SPLINE
SPL {X  -162.820, Y  +574.443, Z    +0.000, E1   +42.333, E3 +366187.799}
SPL {X  -162.820, Y  +568.554, Z    +0.000, E1   +42.362, E3 +366201.161}
SPL {X  -162.820, Y  +561.474, Z    +0.000, E1   +42.369, E3 +366217.346}
SPL {X  -162.820, Y  +555.861, Z    +0.000, E1   +42.349, E3 +366230.151}
SPL {X  -162.820, Y  +550.633, Z    +0.000, E1   +42.421, E3 +366241.681}
SPL {X  -162.820, Y  +546.534, Z    +0.000, E1   +42.268, E3 +366251.890}
SPL {X  -162.820, Y  +539.632, Z    +0.000, E1   +42.488, E3 +366266.611}
SPL {X  -162.820, Y  +533.959, Z    +0.000, E1   +42.310, E3 +366280.308}
SPL {X  -162.820, Y  +527.661, Z    +0.000, E1   +42.425, E3 +366294.304}
SPL {X  -162.820, Y  +521.246, Z    +0.000, E1   +42.365, E3 +366309.057}
SPL {X  -162.820, Y  +515.708, Z    +0.000, E1   +42.333, E3 +366322.019}
SPL {X  -162.820, Y  +510.265, Z    +0.000, E1   +42.390, E3 +366333.981}
SPL {X  -162.820, Y  +505.746, Z    +0.000, E1   +42.400, E3 +366344.293}
SPL {X  -162.820, Y  +500.461, Z    +0.000, E1   +42.387, E3 +366356.421}
SPL {X  -162.820, Y  +494.841, Z    +0.000, E1   +42.316, E3 +366369.747}
SPL {X  -162.820, Y  +486.958, Z    +0.000, E1   +42.460, E3 +366387.040}
SPL {X  -162.820, Y  +464.528, Z    +0.000, E1   +47.611, E3 +366403.253}
SPL {X  -162.820, Y  +458.830, Z    +0.000, E1   +46.994, E3 +366417.931}
SPL {X  -162.820, Y  +455.537, Z    +0.000, E1   +45.900, E3 +366430.750}
SPL {X  -162.820, Y  +452.032, Z    +0.000, E1   +45.224, E3 +366441.955}
SPL {X  -162.820, Y  +446.617, Z    +0.000, E1   +44.768, E3 +366456.041}
SPL {X  -162.820, Y  +440.464, Z    +0.000, E1   +44.845, E3 +366468.343}
SPL {X  -162.820, Y  +435.902, Z    +0.000, E1   +44.853, E3 +366477.867}
SPL {X  -162.820, Y  +429.336, Z    +0.000, E1   +44.917, E3 +366491.385}
SPL {X  -162.820, Y  +423.193, Z    +0.000, E1   +44.819, E3 +366504.644}
SPL {X  -162.820, Y  +416.810, Z    +0.000, E1   +44.932, E3 +366517.532}
SPL {X  -162.820, Y  +408.782, Z    +0.000, E1   +44.820, E3 +366534.963}
SPL {X  -162.820, Y  +401.619, Z    +0.000, E1   +44.978, E3 +366548.885}
SPL {X  -162.820, Y  +394.771, Z    +0.000, E1   +44.856, E3 +366564.124}
SPL {X  -162.820, Y  +387.883, Z    +0.000, E1   +44.837, E3 +366578.478}
SPL {X  -162.820, Y  +382.755, Z    +0.000, E1   +44.828, E3 +366589.271}
SPL {X  -162.796, Y  +377.700, Z    +0.000, E1   +44.829, E3 +366599.851}
SPL {X  -162.619, Y  +372.412, Z    +0.000, E1   +44.928, E3 +366610.310}
SPL {X  -162.311, Y  +367.633, Z    +0.000, E1   +44.798, E3 +366621.077}
SPL {X  -161.766, Y  +362.002, Z    +0.000, E1   +44.644, E3 +366633.836}
SPL {X  -161.043, Y  +356.508, Z    +0.000, E1   +44.528, E3 +366645.950}
SPL {X  -160.070, Y  +350.699, Z    +0.000, E1   +44.409, E3 +366658.902}
SPL {X  -158.853, Y  +344.776, Z    +0.000, E1   +44.148, E3 +366672.723}
SPL {X  -157.292, Y  +338.433, Z    +0.000, E1   +43.917, E3 +366687.401}
SPL {X  -155.654, Y  +332.729, Z    +0.000, E1   +43.534, E3 +366701.323}
SPL {X  -154.189, Y  +328.191, Z    +0.000, E1   +43.338, E3 +366711.820}
SPL {X  -149.333, Y  +315.614, Z    +0.000, E1   +46.650, E3 +366719.135}
SPL {X  -142.680, Y  +302.060, Z    +0.000, E1   +42.084, E3 +366785.480}
ENDSPLINE

SPLINE
SPL {X  -151.184, Y  +320.053, Z    +0.000, E1   +32.435, E3 +366852.723}
SPL {X  -158.917, Y  +345.064, Z    +0.000, E1   +21.858, E3 +366854.071}
SPL {X  -161.350, Y  +358.672, Z    +0.000, E1   +15.089, E3 +366856.774}
SPL {X  -162.491, Y  +370.147, Z    +0.000, E1    +8.815, E3 +366859.709}
SPL {X  -162.816, Y  +379.394, Z    +0.000, E1    +3.267, E3 +366859.536}
SPL {X  -162.820, Y  +384.427, Z    +0.000, E1    -0.390, E3 +366860.056}
SPL {X  -162.820, Y  +387.736, Z    +0.000, E1    -3.142, E3 +366859.337}
SPL {X  -162.820, Y  +391.456, Z    +0.000, E1    -6.603, E3 +366860.123}
SPL {X  -162.820, Y  +397.032, Z    +0.000, E1   -12.435, E3 +366859.570}
SPL {X  -162.820, Y  +406.111, Z    +0.000, E1   -22.010, E3 +366860.622}
SPL {X  -162.820, Y  +418.653, Z    +0.000, E1   -36.657, E3 +366854.974}
SPL {X  -162.820, Y  +440.590, Z    +0.000, E1   -50.152, E3 +366860.220}
SPL {X  -162.820, Y  +447.889, Z    +0.000, E1   -43.424, E3 +366891.366}
SPL {X  -162.820, Y  +478.087, Z    +0.000, E1   -45.903, E3 +366936.585}
ENDSPLINE

SPLINE
SPL {X  -162.820, Y  +474.900, Z    +0.000, E1   -42.394, E3 +366950.737}
ENDSPLINE

SPLINE
SPL {X  -162.820, Y  +480.895, Z    +0.000, E1   -42.223, E3 +366965.399}
SPL {X  -162.820, Y  +485.782, Z    +0.000, E1   -42.348, E3 +366975.744}
SPL {X  -162.820, Y  +489.480, Z    +0.000, E1   -42.230, E3 +366984.971}
SPL {X  -162.820, Y  +494.825, Z    +0.000, E1   -42.287, E3 +366996.919}
SPL {X  -162.820, Y  +501.023, Z    +0.000, E1   -42.347, E3 +367010.801}
SPL {X  -162.820, Y  +506.968, Z    +0.000, E1   -42.248, E3 +367024.992}
SPL {X  -162.820, Y  +513.215, Z    +0.000, E1   -42.304, E3 +367038.966}
SPL {X  -162.820, Y  +518.708, Z    +0.000, E1   -42.272, E3 +367051.688}
SPL {X  -162.820, Y  +525.147, Z    +0.000, E1   -42.298, E3 +367066.430}
SPL {X  -162.820, Y  +531.715, Z    +0.000, E1   -42.312, E3 +367081.256}
SPL {X  -162.820, Y  +537.459, Z    +0.000, E1   -42.308, E3 +367094.515}
SPL {X  -162.820, Y  +542.643, Z    +0.000, E1   -42.173, E3 +367107.107}
SPL {X  -162.820, Y  +549.160, Z    +0.000, E1   -42.387, E3 +367120.866}
SPL {X  -162.820, Y  +554.884, Z    +0.000, E1   -42.207, E3 +367134.951}
SPL {X  -162.820, Y  +561.114, Z    +0.000, E1   -42.336, E3 +367148.531}
SPL {X  -162.820, Y  +566.097, Z    +0.000, E1   -42.118, E3 +367161.142}
SPL {X  -162.820, Y  +571.654, Z    +0.000, E1   -42.313, E3 +367172.795}
SPL {X  -162.820, Y  +577.246, Z    +0.000, E1   -42.284, E3 +367185.760}
SPL {X  -162.820, Y  +582.233, Z    +0.000, E1   -42.188, E3 +367197.740}
SPL {X  -162.820, Y  +588.138, Z    +0.000, E1   -42.308, E3 +367210.638}
SPL {X  -162.820, Y  +593.999, Z    +0.000, E1   -42.301, E3 +367224.048}
SPL {X  -162.820, Y  +599.194, Z    +0.000, E1   -42.235, E3 +367236.353}
SPL {X  -162.820, Y  +604.595, Z    +0.000, E1   -42.290, E3 +367248.384}
SPL {X  -162.820, Y  +609.630, Z    +0.000, E1   -42.276, E3 +367260.010}
SPL {X  -162.820, Y  +614.392, Z    +0.000, E1   -42.242, E3 +367271.110}
SPL {X  -162.820, Y  +620.424, Z    +0.000, E1   -42.277, E3 +367284.858}
SPL {X  -162.820, Y  +626.430, Z    +0.000, E1   -42.291, E3 +367298.408}
SPL {X  -162.820, Y  +631.865, Z    +0.000, E1   -42.327, E3 +367310.701}
SPL {X  -162.820, Y  +637.189, Z    +0.000, E1   -42.236, E3 +367323.375}
SPL {X  -162.820, Y  +642.066, Z    +0.000, E1   -42.247, E3 +367334.497}
SPL {X  -162.820, Y  +646.907, Z    +0.000, E1   -42.249, E3 +367345.617}
SPL {X  -162.820, Y  +652.374, Z    +0.000, E1   -42.262, E3 +367358.055}
SPL {X  -162.820, Y  +657.439, Z    +0.000, E1   -42.251, E3 +367369.728}
SPL {X  -162.820, Y  +663.328, Z    +0.000, E1   -42.283, E3 +367383.130}
SPL {X  -162.820, Y  +669.078, Z    +0.000, E1   -42.263, E3 +367396.326}
SPL {X  -162.819, Y  +673.910, Z    +0.000, E1   -42.244, E3 +367407.520}
SPL {X  -162.729, Y  +678.944, Z    +0.000, E1   -42.273, E3 +367418.888}
SPL {X  -162.479, Y  +684.035, Z    +0.000, E1   -42.168, E3 +367431.225}
SPL {X  -162.026, Y  +689.560, Z    +0.000, E1   -42.192, E3 +367443.714}
SPL {X  -161.446, Y  +694.609, Z    +0.000, E1   -42.094, E3 +367455.846}
SPL {X  -160.889, Y  +698.503, Z    +0.000, E1   -41.849, E3 +367466.120}
SPL {X  -160.100, Y  +703.138, Z    +0.000, E1   -41.824, E3 +367476.978}
SPL {X  -158.994, Y  +708.588, Z    +0.000, E1   -41.616, E3 +367490.698}
SPL {X  -157.709, Y  +713.973, Z    +0.000, E1   -41.360, E3 +367504.480}
SPL {X  -156.530, Y  +718.319, Z    +0.000, E1   -41.164, E3 +367515.424}
SPL {X  -155.547, Y  +721.618, Z    +0.000, E1   -40.968, E3 +367524.048}
SPL {X  -151.388, Y  +733.433, Z    +0.000, E1   -44.269, E3 +367531.751}
SPL {X  -144.352, Y  +748.818, Z    +0.000, E1   -40.701, E3 +367600.786}
SPL {X  -143.859, Y  +749.757, Z    +0.000, E1   -39.148, E3 +367628.734}
ENDSPLINE

SPLINE
SPL {X  -159.245, Y  +707.432, Z    +0.000, E1   -21.244, E3 +367660.767}
SPL {X  -162.277, Y  +686.791, Z    +0.000, E1   -10.607, E3 +367662.178}
SPL {X  -162.766, Y  +677.687, Z    +0.000, E1    -5.239, E3 +367664.368}
SPL {X  -162.820, Y  +671.059, Z    +0.000, E1    -0.934, E3 +367664.724}
SPL {X  -162.820, Y  +665.599, Z    +0.000, E1    +3.424, E3 +367665.173}
SPL {X  -162.820, Y  +661.024, Z    +0.000, E1    +7.880, E3 +367664.642}
SPL {X  -162.820, Y  +654.280, Z    +0.000, E1   +14.617, E3 +367665.359}
SPL {X  -162.820, Y  +638.947, Z    +0.000, E1   +31.033, E3 +367663.413}
SPL {X  -162.820, Y  +608.150, Z    +0.000, E1   +43.921, E3 +367689.645}
SPL {X  -162.820, Y  +574.255, Z    +0.000, E1   +46.562, E3 +367739.439}
ENDSPLINE

SPLINE
SPL {X  -162.820, Y  +579.440, Z    +0.000, E1   +42.450, E3 +367752.627}
ENDSPLINE

SPLINE
SPL {X  -162.820, Y  +574.443, Z    +0.000, E1   +42.333, E3 +367764.722}
SPL {X  -162.820, Y  +568.554, Z    +0.000, E1   +42.362, E3 +367778.084}
SPL {X  -162.820, Y  +561.474, Z    +0.000, E1   +42.369, E3 +367794.269}
SPL {X  -162.820, Y  +555.861, Z    +0.000, E1   +42.349, E3 +367807.074}
SPL {X  -162.820, Y  +550.633, Z    +0.000, E1   +42.421, E3 +367818.604}
SPL {X  -162.820, Y  +546.534, Z    +0.000, E1   +42.268, E3 +367828.813}
SPL {X  -162.820, Y  +541.056, Z    +0.000, E1   +42.452, E3 +367840.328}
SPL {X  -162.820, Y  +535.223, Z    +0.000, E1   +42.386, E3 +367854.022}
SPL {X  -162.820, Y  +529.084, Z    +0.000, E1   +42.400, E3 +367867.945}
SPL {X  -162.820, Y  +522.568, Z    +0.000, E1   +42.385, E3 +367882.975}
SPL {X  -162.820, Y  +515.708, Z    +0.000, E1   +42.333, E3 +367898.942}
SPL {X  -162.820, Y  +510.265, Z    +0.000, E1   +42.390, E3 +367910.904}
SPL {X  -162.820, Y  +505.746, Z    +0.000, E1   +42.400, E3 +367921.216}
SPL {X  -162.820, Y  +500.461, Z    +0.000, E1   +42.387, E3 +367933.344}
SPL {X  -162.820, Y  +494.841, Z    +0.000, E1   +42.316, E3 +367946.670}
SPL {X  -162.820, Y  +487.903, Z    +0.000, E1   +42.488, E3 +367961.493}
SPL {X  -162.820, Y  +484.250, Z    +0.000, E1   +42.201, E3 +367971.354}
SPL {X  -162.820, Y  +464.528, Z    +0.000, E1   +47.611, E3 +367980.176}
SPL {X  -162.820, Y  +459.899, Z    +0.000, E1   +47.097, E3 +367992.019}
SPL {X  -162.820, Y  +455.990, Z    +0.000, E1   +46.212, E3 +368005.093}
SPL {X  -162.820, Y  +452.032, Z    +0.000, E1   +45.224, E3 +368018.878}
SPL {X  -162.820, Y  +446.617, Z    +0.000, E1   +44.768, E3 +368032.965}
SPL {X  -162.820, Y  +437.902, Z    +0.000, E1   +44.900, E3 +368050.541}
SPL {X  -162.820, Y  +429.336, Z    +0.000, E1   +44.917, E3 +368068.308}
SPL {X  -162.820, Y  +423.193, Z    +0.000, E1   +44.819, E3 +368081.567}
SPL {X  -162.820, Y  +416.810, Z    +0.000, E1   +44.932, E3 +368094.455}
SPL {X  -162.820, Y  +408.782, Z    +0.000, E1   +44.820, E3 +368111.886}
SPL {X  -162.820, Y  +401.619, Z    +0.000, E1   +44.978, E3 +368125.808}
SPL {X  -162.820, Y  +394.771, Z    +0.000, E1   +44.856, E3 +368141.047}
SPL {X  -162.820, Y  +387.883, Z    +0.000, E1   +44.837, E3 +368155.401}
SPL {X  -162.820, Y  +382.755, Z    +0.000, E1   +44.828, E3 +368166.194}
SPL {X  -162.796, Y  +377.700, Z    +0.000, E1   +44.829, E3 +368176.774}
SPL {X  -162.619, Y  +372.412, Z    +0.000, E1   +44.928, E3 +368187.233}
SPL {X  -162.311, Y  +367.633, Z    +0.000, E1   +44.798, E3 +368198.000}
SPL {X  -161.766, Y  +362.002, Z    +0.000, E1   +44.644, E3 +368210.759}
SPL {X  -161.043, Y  +356.508, Z    +0.000, E1   +44.528, E3 +368222.874}
SPL {X  -160.070, Y  +350.699, Z    +0.000, E1   +44.409, E3 +368235.825}
SPL {X  -158.853, Y  +344.776, Z    +0.000, E1   +44.148, E3 +368249.646}
SPL {X  -157.292, Y  +338.433, Z    +0.000, E1   +43.917, E3 +368264.324}
SPL {X  -155.654, Y  +332.729, Z    +0.000, E1   +43.534, E3 +368278.246}
SPL {X  -154.189, Y  +328.191, Z    +0.000, E1   +43.338, E3 +368288.743}
SPL {X  -149.333, Y  +315.614, Z    +0.000, E1   +46.650, E3 +368296.059}
SPL {X  -142.680, Y  +302.060, Z    +0.000, E1   +42.084, E3 +368362.403}
ENDSPLINE

SPLINE
SPL {X  -151.184, Y  +320.053, Z    +0.000, E1   +32.435, E3 +368429.646}
SPL {X  -158.917, Y  +345.064, Z    +0.000, E1   +21.858, E3 +368430.994}
SPL {X  -161.350, Y  +358.672, Z    +0.000, E1   +15.089, E3 +368433.697}
SPL {X  -162.491, Y  +370.147, Z    +0.000, E1    +8.815, E3 +368436.632}
SPL {X  -162.771, Y  +376.522, Z    +0.000, E1    +5.005, E3 +368436.241}
SPL {X  -162.820, Y  +383.029, Z    +0.000, E1    +0.769, E3 +368436.809}
SPL {X  -162.820, Y  +387.736, Z    +0.000, E1    -3.142, E3 +368436.260}
SPL {X  -162.820, Y  +391.456, Z    +0.000, E1    -6.603, E3 +368437.046}
SPL {X  -162.820, Y  +397.032, Z    +0.000, E1   -12.435, E3 +368436.493}
SPL {X  -162.820, Y  +406.111, Z    +0.000, E1   -22.010, E3 +368437.545}
SPL {X  -162.820, Y  +418.653, Z    +0.000, E1   -36.657, E3 +368431.897}
SPL {X  -162.820, Y  +440.590, Z    +0.000, E1   -50.152, E3 +368437.143}
SPL {X  -162.820, Y  +447.889, Z    +0.000, E1   -43.424, E3 +368468.289}
SPL {X  -162.820, Y  +478.087, Z    +0.000, E1   -45.903, E3 +368513.508}
ENDSPLINE

SPLINE
SPL {X  -162.820, Y  +474.900, Z    +0.000, E1   -42.394, E3 +368527.660}
ENDSPLINE

SPLINE
SPL {X  -162.820, Y  +480.895, Z    +0.000, E1   -42.223, E3 +368542.322}
SPL {X  -162.820, Y  +488.112, Z    +0.000, E1   -42.323, E3 +368558.403}
SPL {X  -162.820, Y  +494.825, Z    +0.000, E1   -42.287, E3 +368573.842}
SPL {X  -162.820, Y  +501.909, Z    +0.000, E1   -42.324, E3 +368590.028}
SPL {X  -162.820, Y  +508.157, Z    +0.000, E1   -42.280, E3 +368604.359}
SPL {X  -162.820, Y  +513.215, Z    +0.000, E1   -42.304, E3 +368615.889}
SPL {X  -162.820, Y  +518.708, Z    +0.000, E1   -42.272, E3 +368628.611}
SPL {X  -162.820, Y  +525.147, Z    +0.000, E1   -42.298, E3 +368643.353}
SPL {X  -162.820, Y  +531.715, Z    +0.000, E1   -42.312, E3 +368658.179}
SPL {X  -162.820, Y  +537.459, Z    +0.000, E1   -42.308, E3 +368671.438}
SPL {X  -162.820, Y  +542.643, Z    +0.000, E1   -42.173, E3 +368684.030}
SPL {X  -162.820, Y  +547.830, Z    +0.000, E1   -42.372, E3 +368694.709}
SPL {X  -162.820, Y  +553.760, Z    +0.000, E1   -42.287, E3 +368708.986}
SPL {X  -162.820, Y  +561.114, Z    +0.000, E1   -42.336, E3 +368725.454}
SPL {X  -162.820, Y  +566.097, Z    +0.000, E1   -42.118, E3 +368738.065}
SPL {X  -162.820, Y  +571.654, Z    +0.000, E1   -42.313, E3 +368749.718}
SPL {X  -162.820, Y  +577.246, Z    +0.000, E1   -42.284, E3 +368762.684}
SPL {X  -162.820, Y  +582.233, Z    +0.000, E1   -42.188, E3 +368774.663}
SPL {X  -162.820, Y  +588.138, Z    +0.000, E1   -42.308, E3 +368787.561}
SPL {X  -162.820, Y  +593.999, Z    +0.000, E1   -42.301, E3 +368800.971}
SPL {X  -162.820, Y  +599.194, Z    +0.000, E1   -42.235, E3 +368813.276}
SPL {X  -162.820, Y  +604.595, Z    +0.000, E1   -42.290, E3 +368825.307}
SPL {X  -162.820, Y  +609.630, Z    +0.000, E1   -42.276, E3 +368836.933}
SPL {X  -162.820, Y  +614.392, Z    +0.000, E1   -42.242, E3 +368848.033}
SPL {X  -162.820, Y  +618.928, Z    +0.000, E1   -42.220, E3 +368858.559}
SPL {X  -162.820, Y  +625.176, Z    +0.000, E1   -42.323, E3 +368872.411}
SPL {X  -162.820, Y  +630.164, Z    +0.000, E1   -42.259, E3 +368884.021}
SPL {X  -162.820, Y  +635.892, Z    +0.000, E1   -42.319, E3 +368897.013}
SPL {X  -162.820, Y  +642.066, Z    +0.000, E1   -42.247, E3 +368911.421}
SPL {X  -162.820, Y  +646.907, Z    +0.000, E1   -42.249, E3 +368922.540}
SPL {X  -162.820, Y  +652.374, Z    +0.000, E1   -42.262, E3 +368934.978}
SPL {X  -162.820, Y  +657.439, Z    +0.000, E1   -42.251, E3 +368946.651}
SPL {X  -162.820, Y  +663.328, Z    +0.000, E1   -42.283, E3 +368960.053}
SPL {X  -162.820, Y  +669.078, Z    +0.000, E1   -42.263, E3 +368973.249}
SPL {X  -162.819, Y  +673.910, Z    +0.000, E1   -42.244, E3 +368984.443}
SPL {X  -162.729, Y  +678.944, Z    +0.000, E1   -42.273, E3 +368995.811}
SPL {X  -162.479, Y  +684.035, Z    +0.000, E1   -42.168, E3 +369008.148}
SPL {X  -162.026, Y  +689.560, Z    +0.000, E1   -42.192, E3 +369020.637}
SPL {X  -161.446, Y  +694.609, Z    +0.000, E1   -42.094, E3 +369032.769}
SPL {X  -160.681, Y  +699.806, Z    +0.000, E1   -41.866, E3 +369046.052}
SPL {X  -159.658, Y  +705.434, Z    +0.000, E1   -41.735, E3 +369059.682}
SPL {X  -158.502, Y  +710.748, Z    +0.000, E1   -41.532, E3 +369073.029}
SPL {X  -157.452, Y  +714.962, Z    +0.000, E1   -41.276, E3 +369084.025}
SPL {X  -156.530, Y  +718.319, Z    +0.000, E1   -41.164, E3 +369092.348}
SPL {X  -155.547, Y  +721.618, Z    +0.000, E1   -40.968, E3 +369100.971}
SPL {X  -151.388, Y  +733.433, Z    +0.000, E1   -44.269, E3 +369108.674}
SPL {X  -144.352, Y  +748.818, Z    +0.000, E1   -40.701, E3 +369177.709}
SPL {X  -143.859, Y  +749.757, Z    +0.000, E1   -39.148, E3 +369205.657}
ENDSPLINE

SPLINE
SPL {X  -159.245, Y  +707.432, Z    +0.000, E1   -21.244, E3 +369237.690}
SPL {X  -162.277, Y  +686.791, Z    +0.000, E1   -10.607, E3 +369239.101}
SPL {X  -162.766, Y  +677.687, Z    +0.000, E1    -5.239, E3 +369241.291}
SPL {X  -162.820, Y  +672.396, Z    +0.000, E1    -1.801, E3 +369242.079}
SPL {X  -162.820, Y  +667.851, Z    +0.000, E1    +1.551, E3 +369241.576}
SPL {X  -162.820, Y  +664.036, Z    +0.000, E1    +4.934, E3 +369242.295}
SPL {X  -162.820, Y  +661.024, Z    +0.000, E1    +7.880, E3 +369241.565}
SPL {X  -162.820, Y  +656.051, Z    +0.000, E1   +12.848, E3 +369242.432}
SPL {X  -162.820, Y  +650.794, Z    +0.000, E1   +18.580, E3 +369241.988}
SPL {X  -162.820, Y  +638.947, Z    +0.000, E1   +31.033, E3 +369240.336}
SPL {X  -162.820, Y  +608.150, Z    +0.000, E1   +43.921, E3 +369266.569}
SPL {X  -162.820, Y  +574.255, Z    +0.000, E1   +46.562, E3 +369316.362}
ENDSPLINE

SPLINE
SPL {X  -162.820, Y  +579.440, Z    +0.000, E1   +42.450, E3 +369329.550}
ENDSPLINE

SPLINE
SPL {X  -162.820, Y  +574.443, Z    +0.000, E1   +42.333, E3 +369341.645}
SPL {X  -162.820, Y  +568.554, Z    +0.000, E1   +42.362, E3 +369355.007}
SPL {X  -162.820, Y  +561.474, Z    +0.000, E1   +42.369, E3 +369371.192}
SPL {X  -162.820, Y  +555.861, Z    +0.000, E1   +42.349, E3 +369383.997}
SPL {X  -162.820, Y  +550.633, Z    +0.000, E1   +42.421, E3 +369395.527}
SPL {X  -162.820, Y  +546.534, Z    +0.000, E1   +42.268, E3 +369405.736}
SPL {X  -162.820, Y  +539.632, Z    +0.000, E1   +42.488, E3 +369420.458}
SPL {X  -162.820, Y  +533.959, Z    +0.000, E1   +42.310, E3 +369434.154}
SPL {X  -162.820, Y  +527.661, Z    +0.000, E1   +42.425, E3 +369448.150}
SPL {X  -162.820, Y  +521.246, Z    +0.000, E1   +42.365, E3 +369462.903}
SPL {X  -162.820, Y  +515.708, Z    +0.000, E1   +42.333, E3 +369475.865}
SPL {X  -162.820, Y  +510.265, Z    +0.000, E1   +42.390, E3 +369487.827}
SPL {X  -162.820, Y  +505.746, Z    +0.000, E1   +42.400, E3 +369498.140}
SPL {X  -162.820, Y  +500.461, Z    +0.000, E1   +42.387, E3 +369510.267}
SPL {X  -162.820, Y  +494.841, Z    +0.000, E1   +42.316, E3 +369523.593}
SPL {X  -162.820, Y  +486.958, Z    +0.000, E1   +42.460, E3 +369540.886}
SPL {X  -162.820, Y  +464.528, Z    +0.000, E1   +47.611, E3 +369557.099}
SPL {X  -162.820, Y  +458.830, Z    +0.000, E1   +46.994, E3 +369571.777}
SPL {X  -162.820, Y  +455.537, Z    +0.000, E1   +45.900, E3 +369584.596}
SPL {X  -162.820, Y  +452.032, Z    +0.000, E1   +45.224, E3 +369595.801}
SPL {X  -162.820, Y  +446.617, Z    +0.000, E1   +44.768, E3 +369609.888}
SPL {X  -162.820, Y  +440.464, Z    +0.000, E1   +44.845, E3 +369622.190}
SPL {X  -162.820, Y  +435.902, Z    +0.000, E1   +44.853, E3 +369631.713}
SPL {X  -162.820, Y  +429.336, Z    +0.000, E1   +44.917, E3 +369645.231}
SPL {X  -162.820, Y  +423.193, Z    +0.000, E1   +44.819, E3 +369658.490}
SPL {X  -162.820, Y  +416.810, Z    +0.000, E1   +44.932, E3 +369671.378}
SPL {X  -162.820, Y  +408.782, Z    +0.000, E1   +44.820, E3 +369688.809}
SPL {X  -162.820, Y  +401.619, Z    +0.000, E1   +44.978, E3 +369702.731}
SPL {X  -162.820, Y  +394.771, Z    +0.000, E1   +44.856, E3 +369717.970}
SPL {X  -162.820, Y  +387.883, Z    +0.000, E1   +44.837, E3 +369732.324}
SPL {X  -162.820, Y  +382.755, Z    +0.000, E1   +44.828, E3 +369743.117}
SPL {X  -162.796, Y  +377.700, Z    +0.000, E1   +44.829, E3 +369753.697}
SPL {X  -162.619, Y  +372.412, Z    +0.000, E1   +44.928, E3 +369764.156}
SPL {X  -162.311, Y  +367.633, Z    +0.000, E1   +44.798, E3 +369774.923}
SPL {X  -161.766, Y  +362.002, Z    +0.000, E1   +44.644, E3 +369787.682}
SPL {X  -161.043, Y  +356.508, Z    +0.000, E1   +44.528, E3 +369799.797}
SPL {X  -160.070, Y  +350.699, Z    +0.000, E1   +44.409, E3 +369812.748}
SPL {X  -158.853, Y  +344.776, Z    +0.000, E1   +44.148, E3 +369826.569}
SPL {X  -157.292, Y  +338.433, Z    +0.000, E1   +43.917, E3 +369841.247}
SPL {X  -155.654, Y  +332.729, Z    +0.000, E1   +43.534, E3 +369855.169}
SPL {X  -154.189, Y  +328.191, Z    +0.000, E1   +43.338, E3 +369865.666}
SPL {X  -149.333, Y  +315.614, Z    +0.000, E1   +46.650, E3 +369872.982}
SPL {X  -142.680, Y  +302.060, Z    +0.000, E1   +42.084, E3 +369939.326}
ENDSPLINE

SPLINE
SPL {X  -151.184, Y  +320.053, Z    +0.000, E1   +32.435, E3 +370006.569}
SPL {X  -158.917, Y  +345.064, Z    +0.000, E1   +21.858, E3 +370007.917}
SPL {X  -161.350, Y  +358.672, Z    +0.000, E1   +15.089, E3 +370010.620}
SPL {X  -162.491, Y  +370.147, Z    +0.000, E1    +8.815, E3 +370013.555}
SPL {X  -162.816, Y  +379.394, Z    +0.000, E1    +3.267, E3 +370013.382}
SPL {X  -162.820, Y  +384.427, Z    +0.000, E1    -0.390, E3 +370013.902}
SPL {X  -162.820, Y  +387.736, Z    +0.000, E1    -3.142, E3 +370013.183}
SPL {X  -162.820, Y  +391.456, Z    +0.000, E1    -6.603, E3 +370013.969}
SPL {X  -162.820, Y  +397.032, Z    +0.000, E1   -12.435, E3 +370013.416}
SPL {X  -162.820, Y  +406.111, Z    +0.000, E1   -22.010, E3 +370014.468}
SPL {X  -162.820, Y  +418.653, Z    +0.000, E1   -36.657, E3 +370008.821}
SPL {X  -162.820, Y  +440.590, Z    +0.000, E1   -50.152, E3 +370014.066}
SPL {X  -162.820, Y  +447.889, Z    +0.000, E1   -43.424, E3 +370045.212}
SPL {X  -162.820, Y  +478.087, Z    +0.000, E1   -45.903, E3 +370090.431}
ENDSPLINE

SPLINE
SPL {X  -162.820, Y  +472.818, Z    +0.000, E1   -42.437, E3 +370099.372}
ENDSPLINE

SPLINE
SPL {X  -162.820, Y  +476.137, Z    +0.000, E1   -42.304, E3 +370107.786}
SPL {X  -162.820, Y  +480.895, Z    +0.000, E1   -42.223, E3 +370119.245}
SPL {X  -162.820, Y  +488.112, Z    +0.000, E1   -42.323, E3 +370135.326}
SPL {X  -162.820, Y  +496.300, Z    +0.000, E1   -42.332, E3 +370154.038}
SPL {X  -162.820, Y  +503.162, Z    +0.000, E1   -42.272, E3 +370169.955}
SPL {X  -162.820, Y  +508.157, Z    +0.000, E1   -42.280, E3 +370181.282}
SPL {X  -162.820, Y  +513.215, Z    +0.000, E1   -42.304, E3 +370192.812}
SPL {X  -162.820, Y  +520.311, Z    +0.000, E1   -42.317, E3 +370209.111}
SPL {X  -162.820, Y  +526.529, Z    +0.000, E1   -42.247, E3 +370223.580}
SPL {X  -162.820, Y  +532.723, Z    +0.000, E1   -42.344, E3 +370237.322}
SPL {X  -162.820, Y  +538.500, Z    +0.000, E1   -42.256, E3 +370250.943}
SPL {X  -162.820, Y  +542.643, Z    +0.000, E1   -42.173, E3 +370260.953}
SPL {X  -162.820, Y  +549.160, Z    +0.000, E1   -42.387, E3 +370274.712}
SPL {X  -162.820, Y  +554.884, Z    +0.000, E1   -42.207, E3 +370288.798}
SPL {X  -162.820, Y  +561.114, Z    +0.000, E1   -42.336, E3 +370302.378}
SPL {X  -162.820, Y  +566.097, Z    +0.000, E1   -42.118, E3 +370314.988}
SPL {X  -162.820, Y  +571.654, Z    +0.000, E1   -42.313, E3 +370326.641}
SPL {X  -162.820, Y  +577.246, Z    +0.000, E1   -42.284, E3 +370339.607}
SPL {X  -162.820, Y  +582.233, Z    +0.000, E1   -42.188, E3 +370351.586}
SPL {X  -162.820, Y  +588.138, Z    +0.000, E1   -42.308, E3 +370364.484}
SPL {X  -162.820, Y  +593.999, Z    +0.000, E1   -42.301, E3 +370377.894}
SPL {X  -162.820, Y  +599.194, Z    +0.000, E1   -42.235, E3 +370390.199}
SPL {X  -162.820, Y  +604.595, Z    +0.000, E1   -42.290, E3 +370402.230}
SPL {X  -162.820, Y  +609.630, Z    +0.000, E1   -42.276, E3 +370413.856}
SPL {X  -162.820, Y  +614.392, Z    +0.000, E1   -42.242, E3 +370424.956}
SPL {X  -162.820, Y  +620.424, Z    +0.000, E1   -42.277, E3 +370438.704}
SPL {X  -162.820, Y  +628.013, Z    +0.000, E1   -42.320, E3 +370455.876}
SPL {X  -162.820, Y  +635.892, Z    +0.000, E1   -42.319, E3 +370473.936}
SPL {X  -162.820, Y  +642.066, Z    +0.000, E1   -42.247, E3 +370488.344}
SPL {X  -162.820, Y  +646.907, Z    +0.000, E1   -42.249, E3 +370499.463}
SPL {X  -162.820, Y  +652.374, Z    +0.000, E1   -42.262, E3 +370511.901}
SPL {X  -162.820, Y  +657.439, Z    +0.000, E1   -42.251, E3 +370523.574}
SPL {X  -162.820, Y  +663.328, Z    +0.000, E1   -42.283, E3 +370536.976}
SPL {X  -162.820, Y  +669.078, Z    +0.000, E1   -42.263, E3 +370550.172}
SPL {X  -162.819, Y  +673.910, Z    +0.000, E1   -42.244, E3 +370561.366}
SPL {X  -162.729, Y  +678.944, Z    +0.000, E1   -42.273, E3 +370572.734}
SPL {X  -162.479, Y  +684.035, Z    +0.000, E1   -42.168, E3 +370585.071}
SPL {X  -162.026, Y  +689.560, Z    +0.000, E1   -42.192, E3 +370597.560}
SPL {X  -161.446, Y  +694.609, Z    +0.000, E1   -42.094, E3 +370609.692}
SPL {X  -160.889, Y  +698.503, Z    +0.000, E1   -41.849, E3 +370619.966}
SPL {X  -160.100, Y  +703.138, Z    +0.000, E1   -41.824, E3 +370630.824}
SPL {X  -158.994, Y  +708.588, Z    +0.000, E1   -41.616, E3 +370644.544}
SPL {X  -157.709, Y  +713.973, Z    +0.000, E1   -41.360, E3 +370658.326}
SPL {X  -156.530, Y  +718.319, Z    +0.000, E1   -41.164, E3 +370669.271}
SPL {X  -155.547, Y  +721.618, Z    +0.000, E1   -40.968, E3 +370677.894}
SPL {X  -151.388, Y  +733.433, Z    +0.000, E1   -44.269, E3 +370685.597}
SPL {X  -144.352, Y  +748.818, Z    +0.000, E1   -40.701, E3 +370754.632}
SPL {X  -143.859, Y  +749.757, Z    +0.000, E1   -39.148, E3 +370782.580}
ENDSPLINE

SPLINE
SPL {X  -159.245, Y  +707.432, Z    +0.000, E1   -21.244, E3 +370814.614}
SPL {X  -162.277, Y  +686.791, Z    +0.000, E1   -10.607, E3 +370816.024}
SPL {X  -162.766, Y  +677.687, Z    +0.000, E1    -5.239, E3 +370818.214}
SPL {X  -162.820, Y  +672.396, Z    +0.000, E1    -1.801, E3 +370819.002}
SPL {X  -162.820, Y  +667.851, Z    +0.000, E1    +1.551, E3 +370818.499}
SPL {X  -162.820, Y  +662.610, Z    +0.000, E1    +6.209, E3 +370818.873}
SPL {X  -162.820, Y  +654.280, Z    +0.000, E1   +14.617, E3 +370819.206}
SPL {X  -162.820, Y  +638.947, Z    +0.000, E1   +31.033, E3 +370817.259}
SPL {X  -162.820, Y  +608.150, Z    +0.000, E1   +43.921, E3 +370843.492}
SPL {X  -162.820, Y  +574.255, Z    +0.000, E1   +46.562, E3 +370893.286}
ENDSPLINE

SPLINE
SPL {X  -162.820, Y  +579.440, Z    +0.000, E1   +42.450, E3 +370906.473}
ENDSPLINE

SPLINE
SPL {X  -162.820, Y  +573.350, Z    +0.000, E1   +42.340, E3 +370921.151}
SPL {X  -162.820, Y  +565.899, Z    +0.000, E1   +42.413, E3 +370937.734}
SPL {X  -162.820, Y  +560.278, Z    +0.000, E1   +42.308, E3 +370951.072}
SPL {X  -162.820, Y  +555.861, Z    +0.000, E1   +42.349, E3 +370960.920}
SPL {X  -162.820, Y  +550.633, Z    +0.000, E1   +42.421, E3 +370972.450}
SPL {X  -162.820, Y  +546.534, Z    +0.000, E1   +42.268, E3 +370982.659}
SPL {X  -162.820, Y  +539.632, Z    +0.000, E1   +42.488, E3 +370997.381}
SPL {X  -162.820, Y  +533.959, Z    +0.000, E1   +42.310, E3 +371011.077}
SPL {X  -162.820, Y  +527.661, Z    +0.000, E1   +42.425, E3 +371025.073}
SPL {X  -162.820, Y  +521.246, Z    +0.000, E1   +42.365, E3 +371039.826}
SPL {X  -162.820, Y  +515.708, Z    +0.000, E1   +42.333, E3 +371052.788}
SPL {X  -162.820, Y  +510.265, Z    +0.000, E1   +42.390, E3 +371064.750}
SPL {X  -162.820, Y  +505.746, Z    +0.000, E1   +42.400, E3 +371075.063}
SPL {X  -162.820, Y  +500.461, Z    +0.000, E1   +42.387, E3 +371087.190}
SPL {X  -162.820, Y  +494.841, Z    +0.000, E1   +42.316, E3 +371100.516}
SPL {X  -162.820, Y  +486.958, Z    +0.000, E1   +42.460, E3 +371117.809}
SPL {X  -162.820, Y  +464.528, Z    +0.000, E1   +47.611, E3 +371134.022}
SPL {X  -162.820, Y  +459.899, Z    +0.000, E1   +47.097, E3 +371145.865}
SPL {X  -162.820, Y  +455.990, Z    +0.000, E1   +46.212, E3 +371158.939}
SPL {X  -162.820, Y  +452.032, Z    +0.000, E1   +45.224, E3 +371172.724}
SPL {X  -162.820, Y  +446.617, Z    +0.000, E1   +44.768, E3 +371186.811}
SPL {X  -162.820, Y  +437.902, Z    +0.000, E1   +44.900, E3 +371204.388}
SPL {X  -162.820, Y  +430.894, Z    +0.000, E1   +44.976, E3 +371218.373}
SPL {X  -162.820, Y  +425.053, Z    +0.000, E1   +44.824, E3 +371231.635}
SPL {X  -162.820, Y  +418.403, Z    +0.000, E1   +44.941, E3 +371244.748}
SPL {X  -162.820, Y  +412.479, Z    +0.000, E1   +44.780, E3 +371258.179}
SPL {X  -162.820, Y  +406.707, Z    +0.000, E1   +44.849, E3 +371269.751}
SPL {X  -162.820, Y  +401.619, Z    +0.000, E1   +44.978, E3 +371279.654}
SPL {X  -162.820, Y  +394.771, Z    +0.000, E1   +44.856, E3 +371294.893}
SPL {X  -162.820, Y  +387.883, Z    +0.000, E1   +44.837, E3 +371309.247}
SPL {X  -162.820, Y  +382.755, Z    +0.000, E1   +44.828, E3 +371320.040}
SPL {X  -162.796, Y  +377.700, Z    +0.000, E1   +44.829, E3 +371330.620}
SPL {X  -162.619, Y  +372.412, Z    +0.000, E1   +44.928, E3 +371341.079}
SPL {X  -162.311, Y  +367.633, Z    +0.000, E1   +44.798, E3 +371351.846}
SPL {X  -161.766, Y  +362.002, Z    +0.000, E1   +44.644, E3 +371364.605}
SPL {X  -161.043, Y  +356.508, Z    +0.000, E1   +44.528, E3 +371376.720}
SPL {X  -160.070, Y  +350.699, Z    +0.000, E1   +44.409, E3 +371389.672}
SPL {X  -158.853, Y  +344.776, Z    +0.000, E1   +44.148, E3 +371403.492}
SPL {X  -157.821, Y  +340.466, Z    +0.000, E1   +44.026, E3 +371413.085}
SPL {X  -156.950, Y  +337.174, Z    +0.000, E1   +43.768, E3 +371421.450}
SPL {X  -155.654, Y  +332.729, Z    +0.000, E1   +43.534, E3 +371432.092}
SPL {X  -154.189, Y  +328.191, Z    +0.000, E1   +43.338, E3 +371442.589}
SPL {X  -149.333, Y  +315.614, Z    +0.000, E1   +46.650, E3 +371449.905}
SPL {X  -142.680, Y  +302.060, Z    +0.000, E1   +42.084, E3 +371516.249}
ENDSPLINE

SPLINE
SPL {X  -151.184, Y  +320.053, Z    +0.000, E1   +32.435, E3 +371583.492}
SPL {X  -158.917, Y  +345.064, Z    +0.000, E1   +21.858, E3 +371584.840}
SPL {X  -161.350, Y  +358.672, Z    +0.000, E1   +15.089, E3 +371587.543}
SPL {X  -162.491, Y  +370.147, Z    +0.000, E1    +8.815, E3 +371590.478}
SPL {X  -162.816, Y  +379.394, Z    +0.000, E1    +3.267, E3 +371590.306}
SPL {X  -162.820, Y  +384.427, Z    +0.000, E1    -0.390, E3 +371590.825}
SPL {X  -162.820, Y  +387.736, Z    +0.000, E1    -3.142, E3 +371590.106}
SPL {X  -162.820, Y  +391.456, Z    +0.000, E1    -6.603, E3 +371590.892}
SPL {X  -162.820, Y  +397.032, Z    +0.000, E1   -12.435, E3 +371590.339}
SPL {X  -162.820, Y  +406.111, Z    +0.000, E1   -22.010, E3 +371591.391}
SPL {X  -162.820, Y  +418.653, Z    +0.000, E1   -36.657, E3 +371585.744}
SPL {X  -162.820, Y  +440.590, Z    +0.000, E1   -50.152, E3 +371590.989}
SPL {X  -162.820, Y  +447.889, Z    +0.000, E1   -43.424, E3 +371622.135}
SPL {X  -162.820, Y  +478.087, Z    +0.000, E1   -45.903, E3 +371667.354}
ENDSPLINE

SPLINE
SPL {X  -162.820, Y  +472.818, Z    +0.000, E1   -42.437, E3 +371676.295}
ENDSPLINE

SPLINE
SPL {X  -162.820, Y  +477.319, Z    +0.000, E1   -42.306, E3 +371687.521}
SPL {X  -162.820, Y  +483.923, Z    +0.000, E1   -42.291, E3 +371702.728}
SPL {X  -162.820, Y  +489.480, Z    +0.000, E1   -42.230, E3 +371715.741}
SPL {X  -162.820, Y  +494.825, Z    +0.000, E1   -42.287, E3 +371727.688}
SPL {X  -162.820, Y  +501.023, Z    +0.000, E1   -42.347, E3 +371741.570}
SPL {X  -162.820, Y  +506.968, Z    +0.000, E1   -42.248, E3 +371755.761}
SPL {X  -162.820, Y  +513.215, Z    +0.000, E1   -42.304, E3 +371769.735}
SPL {X  -162.820, Y  +518.708, Z    +0.000, E1   -42.272, E3 +371782.457}
SPL {X  -162.820, Y  +525.147, Z    +0.000, E1   -42.298, E3 +371797.199}
SPL {X  -162.820, Y  +531.715, Z    +0.000, E1   -42.312, E3 +371812.025}
SPL {X  -162.820, Y  +537.459, Z    +0.000, E1   -42.308, E3 +371825.284}
SPL {X  -162.820, Y  +542.643, Z    +0.000, E1   -42.173, E3 +371837.876}
SPL {X  -162.820, Y  +549.160, Z    +0.000, E1   -42.387, E3 +371851.635}
SPL {X  -162.820, Y  +554.884, Z    +0.000, E1   -42.207, E3 +371865.721}
SPL {X  -162.820, Y  +561.114, Z    +0.000, E1   -42.336, E3 +371879.301}
SPL {X  -162.820, Y  +566.097, Z    +0.000, E1   -42.118, E3 +371891.911}
SPL {X  -162.820, Y  +571.654, Z    +0.000, E1   -42.313, E3 +371903.564}
SPL {X  -162.820, Y  +577.246, Z    +0.000, E1   -42.284, E3 +371916.530}
SPL {X  -162.820, Y  +583.926, Z    +0.000, E1   -42.266, E3 +371932.089}
SPL {X  -162.820, Y  +589.581, Z    +0.000, E1   -42.277, E3 +371944.767}
SPL {X  -162.820, Y  +593.999, Z    +0.000, E1   -42.301, E3 +371954.817}
SPL {X  -162.820, Y  +599.194, Z    +0.000, E1   -42.235, E3 +371967.122}
SPL {X  -162.820, Y  +604.595, Z    +0.000, E1   -42.290, E3 +371979.153}
SPL {X  -162.820, Y  +609.630, Z    +0.000, E1   -42.276, E3 +371990.779}
SPL {X  -162.820, Y  +614.392, Z    +0.000, E1   -42.242, E3 +372001.879}
SPL {X  -162.820, Y  +620.424, Z    +0.000, E1   -42.277, E3 +372015.627}
SPL {X  -162.820, Y  +626.430, Z    +0.000, E1   -42.291, E3 +372029.177}
SPL {X  -162.820, Y  +631.865, Z    +0.000, E1   -42.327, E3 +372041.470}
SPL {X  -162.820, Y  +637.189, Z    +0.000, E1   -42.236, E3 +372054.144}
SPL {X  -162.820, Y  +642.066, Z    +0.000, E1   -42.247, E3 +372065.267}
SPL {X  -162.820, Y  +646.907, Z    +0.000, E1   -42.249, E3 +372076.386}
SPL {X  -162.820, Y  +652.374, Z    +0.000, E1   -42.262, E3 +372088.824}
SPL {X  -162.820, Y  +657.439, Z    +0.000, E1   -42.251, E3 +372100.497}
SPL {X  -162.820, Y  +663.328, Z    +0.000, E1   -42.283, E3 +372113.899}
SPL {X  -162.820, Y  +669.078, Z    +0.000, E1   -42.263, E3 +372127.095}
SPL {X  -162.819, Y  +673.910, Z    +0.000, E1   -42.244, E3 +372138.289}
SPL {X  -162.729, Y  +678.944, Z    +0.000, E1   -42.273, E3 +372149.657}
SPL {X  -162.479, Y  +684.035, Z    +0.000, E1   -42.168, E3 +372161.994}
SPL {X  -162.026, Y  +689.560, Z    +0.000, E1   -42.192, E3 +372174.483}
SPL {X  -161.446, Y  +694.609, Z    +0.000, E1   -42.094, E3 +372186.615}
SPL {X  -160.889, Y  +698.503, Z    +0.000, E1   -41.849, E3 +372196.889}
SPL {X  -159.869, Y  +704.360, Z    +0.000, E1   -41.806, E3 +372210.830}
SPL {X  -158.502, Y  +710.748, Z    +0.000, E1   -41.532, E3 +372226.875}
SPL {X  -156.963, Y  +716.777, Z    +0.000, E1   -41.265, E3 +372242.298}
SPL {X  -155.547, Y  +721.618, Z    +0.000, E1   -40.968, E3 +372254.818}
SPL {X  -151.388, Y  +733.433, Z    +0.000, E1   -44.269, E3 +372262.520}
SPL {X  -144.352, Y  +748.818, Z    +0.000, E1   -40.701, E3 +372331.555}
SPL {X  -143.859, Y  +749.757, Z    +0.000, E1   -39.148, E3 +372359.503}
ENDSPLINE

SPLINE
SPL {X  -159.245, Y  +707.432, Z    +0.000, E1   -21.244, E3 +372391.537}
SPL {X  -162.277, Y  +686.791, Z    +0.000, E1   -10.607, E3 +372392.947}
SPL {X  -162.766, Y  +677.687, Z    +0.000, E1    -5.239, E3 +372395.137}
SPL {X  -162.820, Y  +672.396, Z    +0.000, E1    -1.801, E3 +372395.925}
SPL {X  -162.820, Y  +667.851, Z    +0.000, E1    +1.551, E3 +372395.422}
SPL {X  -162.820, Y  +662.610, Z    +0.000, E1    +6.209, E3 +372395.796}
SPL {X  -162.820, Y  +654.280, Z    +0.000, E1   +14.617, E3 +372396.129}
SPL {X  -162.820, Y  +638.947, Z    +0.000, E1   +31.033, E3 +372394.182}
SPL {X  -162.820, Y  +608.150, Z    +0.000, E1   +43.921, E3 +372420.415}
SPL {X  -162.820, Y  +574.255, Z    +0.000, E1   +46.562, E3 +372470.209}
ENDSPLINE

SPLINE
SPL {X  -162.820, Y  +579.440, Z    +0.000, E1   +42.450, E3 +372483.396}
ENDSPLINE

SPLINE
SPL {X  -162.820, Y  +574.443, Z    +0.000, E1   +42.333, E3 +372495.491}
SPL {X  -162.820, Y  +568.554, Z    +0.000, E1   +42.362, E3 +372508.853}
SPL {X  -162.820, Y  +563.699, Z    +0.000, E1   +42.375, E3 +372519.710}
SPL {X  -162.820, Y  +560.278, Z    +0.000, E1   +42.308, E3 +372527.995}
SPL {X  -162.820, Y  +554.421, Z    +0.000, E1   +42.414, E3 +372540.863}
SPL {X  -162.820, Y  +547.774, Z    +0.000, E1   +42.344, E3 +372556.436}
SPL {X  -162.820, Y  +541.056, Z    +0.000, E1   +42.452, E3 +372571.098}
SPL {X  -162.820, Y  +535.223, Z    +0.000, E1   +42.386, E3 +372584.791}
SPL {X  -162.820, Y  +529.084, Z    +0.000, E1   +42.400, E3 +372598.714}
SPL {X  -162.820, Y  +524.911, Z    +0.000, E1   +42.325, E3 +372608.560}
SPL {X  -162.820, Y  +519.984, Z    +0.000, E1   +42.385, E3 +372619.631}
SPL {X  -162.820, Y  +514.684, Z    +0.000, E1   +42.289, E3 +372632.202}
SPL {X  -162.820, Y  +508.859, Z    +0.000, E1   +42.416, E3 +372644.853}
SPL {X  -162.820, Y  +501.651, Z    +0.000, E1   +42.423, E3 +372661.329}
SPL {X  -162.820, Y  +496.578, Z    +0.000, E1   +42.329, E3 +372673.237}
SPL {X  -162.820, Y  +493.739, Z    +0.000, E1   +42.260, E3 +372680.176}
SPL {X  -162.820, Y  +487.903, Z    +0.000, E1   +42.488, E3 +372692.262}
SPL {X  -162.820, Y  +484.250, Z    +0.000, E1   +42.201, E3 +372702.123}
SPL {X  -162.820, Y  +464.528, Z    +0.000, E1   +47.611, E3 +372710.946}
SPL {X  -162.820, Y  +459.899, Z    +0.000, E1   +47.097, E3 +372722.788}
SPL {X  -162.820, Y  +455.990, Z    +0.000, E1   +46.212, E3 +372735.862}
SPL {X  -162.820, Y  +451.000, Z    +0.000, E1   +45.084, E3 +372752.817}
SPL {X  -162.820, Y  +442.850, Z    +0.000, E1   +44.856, E3 +372771.194}
SPL {X  -162.820, Y  +435.902, Z    +0.000, E1   +44.853, E3 +372785.559}
SPL {X  -162.820, Y  +429.336, Z    +0.000, E1   +44.917, E3 +372799.078}
SPL {X  -162.820, Y  +423.193, Z    +0.000, E1   +44.819, E3 +372812.337}
SPL {X  -162.820, Y  +418.403, Z    +0.000, E1   +44.941, E3 +372821.671}
SPL {X  -162.820, Y  +412.479, Z    +0.000, E1   +44.780, E3 +372835.102}
SPL {X  -162.820, Y  +406.707, Z    +0.000, E1   +44.849, E3 +372846.674}
SPL {X  -162.820, Y  +400.166, Z    +0.000, E1   +44.948, E3 +372859.959}
SPL {X  -162.820, Y  +393.279, Z    +0.000, E1   +44.825, E3 +372874.961}
SPL {X  -162.820, Y  +387.883, Z    +0.000, E1   +44.837, E3 +372886.170}
SPL {X  -162.820, Y  +382.755, Z    +0.000, E1   +44.828, E3 +372896.963}
SPL {X  -162.796, Y  +377.700, Z    +0.000, E1   +44.829, E3 +372907.543}
SPL {X  -162.619, Y  +372.412, Z    +0.000, E1   +44.928, E3 +372918.002}
SPL {X  -162.311, Y  +367.633, Z    +0.000, E1   +44.798, E3 +372928.769}
SPL {X  -161.766, Y  +362.002, Z    +0.000, E1   +44.644, E3 +372941.528}
SPL {X  -161.043, Y  +356.508, Z    +0.000, E1   +44.528, E3 +372953.643}
SPL {X  -160.070, Y  +350.699, Z    +0.000, E1   +44.409, E3 +372966.595}
SPL {X  -158.853, Y  +344.776, Z    +0.000, E1   +44.148, E3 +372980.415}
SPL {X  -157.821, Y  +340.466, Z    +0.000, E1   +44.026, E3 +372990.008}
SPL {X  -156.950, Y  +337.174, Z    +0.000, E1   +43.768, E3 +372998.374}
SPL {X  -155.654, Y  +332.729, Z    +0.000, E1   +43.534, E3 +373009.015}
SPL {X  -154.189, Y  +328.191, Z    +0.000, E1   +43.338, E3 +373019.512}
SPL {X  -149.333, Y  +315.614, Z    +0.000, E1   +46.650, E3 +373026.828}
SPL {X  -142.680, Y  +302.060, Z    +0.000, E1   +42.084, E3 +373093.172}
ENDSPLINE

SPLINE
SPL {X  -151.184, Y  +320.053, Z    +0.000, E1   +32.435, E3 +373160.415}
SPL {X  -158.917, Y  +345.064, Z    +0.000, E1   +21.858, E3 +373161.763}
SPL {X  -161.350, Y  +358.672, Z    +0.000, E1   +15.089, E3 +373164.466}
SPL {X  -162.491, Y  +370.147, Z    +0.000, E1    +8.815, E3 +373167.401}
SPL {X  -162.771, Y  +376.522, Z    +0.000, E1    +5.005, E3 +373167.010}
SPL {X  -162.820, Y  +381.116, Z    +0.000, E1    +2.017, E3 +373167.344}
SPL {X  -162.820, Y  +384.427, Z    +0.000, E1    -0.390, E3 +373167.748}
SPL {X  -162.820, Y  +387.736, Z    +0.000, E1    -3.142, E3 +373167.029}
SPL {X  -162.820, Y  +391.456, Z    +0.000, E1    -6.603, E3 +373167.816}
SPL {X  -162.820, Y  +397.032, Z    +0.000, E1   -12.435, E3 +373167.263}
SPL {X  -162.820, Y  +406.111, Z    +0.000, E1   -22.010, E3 +373168.314}
SPL {X  -162.820, Y  +418.653, Z    +0.000, E1   -36.657, E3 +373162.667}
SPL {X  -162.820, Y  +440.590, Z    +0.000, E1   -50.152, E3 +373167.912}
SPL {X  -162.820, Y  +447.889, Z    +0.000, E1   -43.424, E3 +373199.058}
SPL {X  -162.820, Y  +478.087, Z    +0.000, E1   -45.903, E3 +373244.277}
ENDSPLINE

SPLINE
SPL {X  -162.820, Y  +472.818, Z    +0.000, E1   -42.437, E3 +373253.218}
ENDSPLINE

SPLINE
SPL {X  -162.820, Y  +477.319, Z    +0.000, E1   -42.306, E3 +373264.444}
SPL {X  -162.820, Y  +483.923, Z    +0.000, E1   -42.291, E3 +373279.651}
SPL {X  -162.820, Y  +489.480, Z    +0.000, E1   -42.230, E3 +373292.664}
SPL {X  -162.820, Y  +494.825, Z    +0.000, E1   -42.287, E3 +373304.611}
SPL {X  -162.820, Y  +501.023, Z    +0.000, E1   -42.347, E3 +373318.493}
SPL {X  -162.820, Y  +506.968, Z    +0.000, E1   -42.248, E3 +373332.684}
SPL {X  -162.820, Y  +513.215, Z    +0.000, E1   -42.304, E3 +373346.658}
SPL {X  -162.820, Y  +518.708, Z    +0.000, E1   -42.272, E3 +373359.380}
SPL {X  -162.820, Y  +525.147, Z    +0.000, E1   -42.298, E3 +373374.122}
SPL {X  -162.820, Y  +531.715, Z    +0.000, E1   -42.312, E3 +373388.948}
SPL {X  -162.820, Y  +537.459, Z    +0.000, E1   -42.308, E3 +373402.207}
SPL {X  -162.820, Y  +542.643, Z    +0.000, E1   -42.173, E3 +373414.799}
SPL {X  -162.820, Y  +549.160, Z    +0.000, E1   -42.387, E3 +373428.558}
SPL {X  -162.820, Y  +554.884, Z    +0.000, E1   -42.207, E3 +373442.644}
SPL {X  -162.820, Y  +559.897, Z    +0.000, E1   -42.319, E3 +373453.429}
SPL {X  -162.820, Y  +565.154, Z    +0.000, E1   -42.205, E3 +373466.275}
SPL {X  -162.820, Y  +571.654, Z    +0.000, E1   -42.313, E3 +373480.487}
SPL {X  -162.820, Y  +577.246, Z    +0.000, E1   -42.284, E3 +373493.453}
SPL {X  -162.820, Y  +582.233, Z    +0.000, E1   -42.188, E3 +373505.432}
SPL {X  -162.820, Y  +588.138, Z    +0.000, E1   -42.308, E3 +373518.330}
SPL {X  -162.820, Y  +593.999, Z    +0.000, E1   -42.301, E3 +373531.740}
SPL {X  -162.820, Y  +599.194, Z    +0.000, E1   -42.235, E3 +373544.045}
SPL {X  -162.820, Y  +604.595, Z    +0.000, E1   -42.290, E3 +373556.076}
SPL {X  -162.820, Y  +609.630, Z    +0.000, E1   -42.276, E3 +373567.702}
SPL {X  -162.820, Y  +614.392, Z    +0.000, E1   -42.242, E3 +373578.802}
SPL {X  -162.820, Y  +618.928, Z    +0.000, E1   -42.220, E3 +373589.328}
SPL {X  -162.820, Y  +625.176, Z    +0.000, E1   -42.323, E3 +373603.180}
SPL {X  -162.820, Y  +630.164, Z    +0.000, E1   -42.259, E3 +373614.790}
SPL {X  -162.820, Y  +635.892, Z    +0.000, E1   -42.319, E3 +373627.782}
SPL {X  -162.820, Y  +642.066, Z    +0.000, E1   -42.247, E3 +373642.190}
SPL {X  -162.820, Y  +646.907, Z    +0.000, E1   -42.249, E3 +373653.309}
SPL {X  -162.820, Y  +652.374, Z    +0.000, E1   -42.262, E3 +373665.747}
SPL {X  -162.820, Y  +657.439, Z    +0.000, E1   -42.251, E3 +373677.420}
SPL {X  -162.820, Y  +663.328, Z    +0.000, E1   -42.283, E3 +373690.822}
SPL {X  -162.820, Y  +669.078, Z    +0.000, E1   -42.263, E3 +373704.018}
SPL {X  -162.819, Y  +673.910, Z    +0.000, E1   -42.244, E3 +373715.212}
SPL {X  -162.729, Y  +678.944, Z    +0.000, E1   -42.273, E3 +373726.580}
SPL {X  -162.479, Y  +684.035, Z    +0.000, E1   -42.168, E3 +373738.917}
SPL {X  -162.026, Y  +689.560, Z    +0.000, E1   -42.192, E3 +373751.406}
SPL {X  -161.446, Y  +694.609, Z    +0.000, E1   -42.094, E3 +373763.538}
SPL {X  -160.889, Y  +698.503, Z    +0.000, E1   -41.849, E3 +373773.812}
SPL {X  -159.869, Y  +704.360, Z    +0.000, E1   -41.806, E3 +373787.753}
SPL {X  -158.502, Y  +710.748, Z    +0.000, E1   -41.532, E3 +373803.798}
SPL {X  -156.963, Y  +716.777, Z    +0.000, E1   -41.265, E3 +373819.221}
SPL {X  -155.547, Y  +721.618, Z    +0.000, E1   -40.968, E3 +373831.741}
SPL {X  -151.388, Y  +733.433, Z    +0.000, E1   -44.269, E3 +373839.443}
SPL {X  -144.352, Y  +748.818, Z    +0.000, E1   -40.701, E3 +373908.478}
SPL {X  -143.859, Y  +749.757, Z    +0.000, E1   -39.148, E3 +373936.426}
ENDSPLINE

SPLINE
SPL {X  -159.245, Y  +707.432, Z    +0.000, E1   -21.244, E3 +373968.460}
SPL {X  -162.277, Y  +686.791, Z    +0.000, E1   -10.607, E3 +373969.870}
SPL {X  -162.766, Y  +677.687, Z    +0.000, E1    -5.239, E3 +373972.060}
SPL {X  -162.820, Y  +672.396, Z    +0.000, E1    -1.801, E3 +373972.848}
SPL {X  -162.820, Y  +667.851, Z    +0.000, E1    +1.551, E3 +373972.345}
SPL {X  -162.820, Y  +662.610, Z    +0.000, E1    +6.209, E3 +373972.719}
SPL {X  -162.820, Y  +654.280, Z    +0.000, E1   +14.617, E3 +373973.052}
SPL {X  -162.820, Y  +638.947, Z    +0.000, E1   +31.033, E3 +373971.105}
SPL {X  -162.820, Y  +608.150, Z    +0.000, E1   +43.921, E3 +373997.338}
SPL {X  -162.820, Y  +574.255, Z    +0.000, E1   +46.562, E3 +374047.132}
ENDSPLINE

SPLINE
SPL {X  -162.820, Y  +579.440, Z    +0.000, E1   +42.450, E3 +374060.319}
ENDSPLINE

SPLINE
SPL {X  -162.820, Y  +573.350, Z    +0.000, E1   +42.340, E3 +374074.997}
SPL {X  -162.820, Y  +565.899, Z    +0.000, E1   +42.413, E3 +374091.580}
SPL {X  -162.820, Y  +560.278, Z    +0.000, E1   +42.308, E3 +374104.918}
SPL {X  -162.820, Y  +555.861, Z    +0.000, E1   +42.349, E3 +374114.766}
SPL {X  -162.820, Y  +550.633, Z    +0.000, E1   +42.421, E3 +374126.296}
SPL {X  -162.820, Y  +546.534, Z    +0.000, E1   +42.268, E3 +374136.505}
SPL {X  -162.820, Y  +539.632, Z    +0.000, E1   +42.488, E3 +374151.227}
SPL {X  -162.820, Y  +533.959, Z    +0.000, E1   +42.310, E3 +374164.924}
SPL {X  -162.820, Y  +527.661, Z    +0.000, E1   +42.425, E3 +374178.919}
SPL {X  -162.820, Y  +521.246, Z    +0.000, E1   +42.365, E3 +374193.672}
SPL {X  -162.820, Y  +515.708, Z    +0.000, E1   +42.333, E3 +374206.634}
SPL {X  -162.820, Y  +510.265, Z    +0.000, E1   +42.390, E3 +374218.596}
SPL {X  -162.820, Y  +505.746, Z    +0.000, E1   +42.400, E3 +374228.909}
SPL {X  -162.820, Y  +500.461, Z    +0.000, E1   +42.387, E3 +374241.036}
SPL {X  -162.820, Y  +494.841, Z    +0.000, E1   +42.316, E3 +374254.362}
SPL {X  -162.820, Y  +486.958, Z    +0.000, E1   +42.460, E3 +374271.655}
SPL {X  -162.820, Y  +464.528, Z    +0.000, E1   +47.611, E3 +374287.869}
SPL {X  -162.820, Y  +459.899, Z    +0.000, E1   +47.097, E3 +374299.711}
SPL {X  -162.820, Y  +455.990, Z    +0.000, E1   +46.212, E3 +374312.785}
SPL {X  -162.820, Y  +452.032, Z    +0.000, E1   +45.224, E3 +374326.570}
SPL {X  -162.820, Y  +446.617, Z    +0.000, E1   +44.768, E3 +374340.657}
SPL {X  -162.820, Y  +437.902, Z    +0.000, E1   +44.900, E3 +374358.234}
SPL {X  -162.820, Y  +430.894, Z    +0.000, E1   +44.976, E3 +374372.219}
SPL {X  -162.820, Y  +425.053, Z    +0.000, E1   +44.824, E3 +374385.481}
SPL {X  -162.820, Y  +418.403, Z    +0.000, E1   +44.941, E3 +374398.595}
SPL {X  -162.820, Y  +412.479, Z    +0.000, E1   +44.780, E3 +374412.025}
SPL {X  -162.820, Y  +406.707, Z    +0.000, E1   +44.849, E3 +374423.597}
SPL {X  -162.820, Y  +401.619, Z    +0.000, E1   +44.978, E3 +374433.500}
SPL {X  -162.820, Y  +394.771, Z    +0.000, E1   +44.856, E3 +374448.739}
SPL {X  -162.820, Y  +387.883, Z    +0.000, E1   +44.837, E3 +374463.093}
SPL {X  -162.820, Y  +382.755, Z    +0.000, E1   +44.828, E3 +374473.886}
SPL {X  -162.796, Y  +377.700, Z    +0.000, E1   +44.829, E3 +374484.466}
SPL {X  -162.619, Y  +372.412, Z    +0.000, E1   +44.928, E3 +374494.925}
SPL {X  -162.311, Y  +367.633, Z    +0.000, E1   +44.798, E3 +374505.693}
SPL {X  -161.766, Y  +362.002, Z    +0.000, E1   +44.644, E3 +374518.451}
SPL {X  -161.043, Y  +356.508, Z    +0.000, E1   +44.528, E3 +374530.566}
SPL {X  -160.070, Y  +350.699, Z    +0.000, E1   +44.409, E3 +374543.518}
SPL {X  -158.853, Y  +344.776, Z    +0.000, E1   +44.148, E3 +374557.338}
SPL {X  -157.821, Y  +340.466, Z    +0.000, E1   +44.026, E3 +374566.931}
SPL {X  -156.950, Y  +337.174, Z    +0.000, E1   +43.768, E3 +374575.297}
SPL {X  -155.654, Y  +332.729, Z    +0.000, E1   +43.534, E3 +374585.938}
SPL {X  -154.189, Y  +328.191, Z    +0.000, E1   +43.338, E3 +374596.435}
SPL {X  -149.333, Y  +315.614, Z    +0.000, E1   +46.650, E3 +374603.751}
SPL {X  -142.680, Y  +302.060, Z    +0.000, E1   +42.084, E3 +374670.095}
ENDSPLINE

SPLINE
SPL {X  -151.184, Y  +320.053, Z    +0.000, E1   +32.435, E3 +374737.338}
SPL {X  -158.917, Y  +345.064, Z    +0.000, E1   +21.858, E3 +374738.687}
SPL {X  -161.350, Y  +358.672, Z    +0.000, E1   +15.089, E3 +374741.389}
SPL {X  -162.491, Y  +370.147, Z    +0.000, E1    +8.815, E3 +374744.324}
SPL {X  -162.771, Y  +376.522, Z    +0.000, E1    +5.005, E3 +374743.933}
SPL {X  -162.820, Y  +383.029, Z    +0.000, E1    +0.769, E3 +374744.501}
SPL {X  -162.820, Y  +387.736, Z    +0.000, E1    -3.142, E3 +374743.952}
SPL {X  -162.820, Y  +392.770, Z    +0.000, E1    -7.830, E3 +374744.604}
SPL {X  -162.820, Y  +398.469, Z    +0.000, E1   -14.078, E3 +374744.057}
SPL {X  -162.820, Y  +406.111, Z    +0.000, E1   -22.010, E3 +374745.237}
SPL {X  -162.820, Y  +418.653, Z    +0.000, E1   -36.657, E3 +374739.590}
SPL {X  -162.820, Y  +440.590, Z    +0.000, E1   -50.152, E3 +374744.835}
SPL {X  -162.820, Y  +447.889, Z    +0.000, E1   -43.424, E3 +374775.981}
SPL {X  -162.820, Y  +479.020, Z    +0.000, E1   -47.189, E3 +374815.557}
ENDSPLINE

SPLINE
SPL {X  -162.820, Y  +474.886, Z    +0.000, E1   -43.721, E3 +374827.442}
ENDSPLINE

SPLINE
SPL {X  -162.820, Y  +476.137, Z    +0.000, E1   -42.304, E3 +374838.555}
SPL {X  -162.820, Y  +480.895, Z    +0.000, E1   -42.223, E3 +374850.014}
SPL {X  -162.820, Y  +485.782, Z    +0.000, E1   -42.348, E3 +374860.360}
SPL {X  -162.820, Y  +489.480, Z    +0.000, E1   -42.230, E3 +374869.587}
SPL {X  -162.820, Y  +496.300, Z    +0.000, E1   -42.332, E3 +374884.808}
SPL {X  -162.820, Y  +503.162, Z    +0.000, E1   -42.272, E3 +374900.724}
SPL {X  -162.820, Y  +509.376, Z    +0.000, E1   -42.304, E3 +374914.815}
SPL {X  -162.820, Y  +514.403, Z    +0.000, E1   -42.285, E3 +374926.311}
SPL {X  -162.820, Y  +518.708, Z    +0.000, E1   -42.272, E3 +374936.303}
SPL {X  -162.820, Y  +525.147, Z    +0.000, E1   -42.298, E3 +374951.045}
SPL {X  -162.820, Y  +531.715, Z    +0.000, E1   -42.312, E3 +374965.871}
SPL {X  -162.820, Y  +537.459, Z    +0.000, E1   -42.308, E3 +374979.130}
SPL {X  -162.820, Y  +542.643, Z    +0.000, E1   -42.173, E3 +374991.723}
SPL {X  -162.820, Y  +549.160, Z    +0.000, E1   -42.387, E3 +375005.481}
SPL {X  -162.820, Y  +554.884, Z    +0.000, E1   -42.207, E3 +375019.567}
SPL {X  -162.820, Y  +559.897, Z    +0.000, E1   -42.319, E3 +375030.352}
SPL {X  -162.820, Y  +565.154, Z    +0.000, E1   -42.205, E3 +375043.198}
SPL {X  -162.820, Y  +571.654, Z    +0.000, E1   -42.313, E3 +375057.410}
SPL {X  -162.820, Y  +577.246, Z    +0.000, E1   -42.284, E3 +375070.376}
SPL {X  -162.820, Y  +582.233, Z    +0.000, E1   -42.188, E3 +375082.355}
SPL {X  -162.820, Y  +588.138, Z    +0.000, E1   -42.308, E3 +375095.253}
SPL {X  -162.820, Y  +593.999, Z    +0.000, E1   -42.301, E3 +375108.663}
SPL {X  -162.820, Y  +599.194, Z    +0.000, E1   -42.235, E3 +375120.968}
SPL {X  -162.820, Y  +604.595, Z    +0.000, E1   -42.290, E3 +375133.000}
SPL {X  -162.820, Y  +609.630, Z    +0.000, E1   -42.276, E3 +375144.625}
SPL {X  -162.820, Y  +614.392, Z    +0.000, E1   -42.242, E3 +375155.726}
SPL {X  -162.820, Y  +620.424, Z    +0.000, E1   -42.277, E3 +375169.473}
SPL {X  -162.820, Y  +626.430, Z    +0.000, E1   -42.291, E3 +375183.023}
SPL {X  -162.820, Y  +631.865, Z    +0.000, E1   -42.327, E3 +375195.317}
SPL {X  -162.820, Y  +637.189, Z    +0.000, E1   -42.236, E3 +375207.991}
SPL {X  -162.820, Y  +642.066, Z    +0.000, E1   -42.247, E3 +375219.113}
SPL {X  -162.820, Y  +646.907, Z    +0.000, E1   -42.249, E3 +375230.232}
SPL {X  -162.820, Y  +652.374, Z    +0.000, E1   -42.262, E3 +375242.670}
SPL {X  -162.820, Y  +658.634, Z    +0.000, E1   -42.281, E3 +375257.027}
SPL {X  -162.820, Y  +664.480, Z    +0.000, E1   -42.257, E3 +375270.422}
SPL {X  -162.820, Y  +669.078, Z    +0.000, E1   -42.263, E3 +375280.941}
SPL {X  -162.819, Y  +673.910, Z    +0.000, E1   -42.244, E3 +375292.136}
SPL {X  -162.670, Y  +680.491, Z    +0.000, E1   -42.282, E3 +375307.178}
SPL {X  -162.151, Y  +688.243, Z    +0.000, E1   -42.207, E3 +375325.379}
SPL {X  -161.446, Y  +694.609, Z    +0.000, E1   -42.094, E3 +375340.461}
SPL {X  -160.681, Y  +699.806, Z    +0.000, E1   -41.866, E3 +375353.744}
SPL {X  -159.658, Y  +705.434, Z    +0.000, E1   -41.735, E3 +375367.374}
SPL {X  -158.727, Y  +709.780, Z    +0.000, E1   -41.560, E3 +375378.241}
SPL {X  -157.709, Y  +713.973, Z    +0.000, E1   -41.360, E3 +375389.095}
SPL {X  -156.530, Y  +718.319, Z    +0.000, E1   -41.164, E3 +375400.040}
SPL {X  -155.547, Y  +721.618, Z    +0.000, E1   -40.968, E3 +375408.664}
SPL {X  -151.388, Y  +733.433, Z    +0.000, E1   -44.269, E3 +375416.366}
SPL {X  -144.352, Y  +748.818, Z    +0.000, E1   -40.701, E3 +375485.401}
SPL {X  -143.859, Y  +749.757, Z    +0.000, E1   -39.148, E3 +375513.350}
ENDSPLINE

SPLINE
SPL {X  -159.245, Y  +707.432, Z    +0.000, E1   -21.244, E3 +375545.383}
SPL {X  -162.277, Y  +686.791, Z    +0.000, E1   -10.607, E3 +375546.793}
SPL {X  -162.766, Y  +677.687, Z    +0.000, E1    -5.239, E3 +375548.983}
SPL {X  -162.820, Y  +671.059, Z    +0.000, E1    -0.934, E3 +375549.339}
SPL {X  -162.820, Y  +666.960, Z    +0.000, E1    +2.343, E3 +375549.616}
SPL {X  -162.820, Y  +662.610, Z    +0.000, E1    +6.209, E3 +375549.642}
SPL {X  -162.820, Y  +654.280, Z    +0.000, E1   +14.617, E3 +375549.975}
SPL {X  -162.820, Y  +638.947, Z    +0.000, E1   +31.033, E3 +375548.028}
SPL {X  -162.820, Y  +608.150, Z    +0.000, E1   +43.921, E3 +375574.261}
SPL {X  -162.820, Y  +574.255, Z    +0.000, E1   +46.562, E3 +375624.055}
ENDSPLINE

SPLINE
SPL {X  -162.820, Y  +579.440, Z    +0.000, E1   +42.450, E3 +375637.242}
ENDSPLINE

SPLINE
SPL {X  -162.820, Y  +574.443, Z    +0.000, E1   +42.333, E3 +375649.337}
SPL {X  -162.820, Y  +568.554, Z    +0.000, E1   +42.362, E3 +375662.699}
SPL {X  -162.820, Y  +561.474, Z    +0.000, E1   +42.369, E3 +375678.885}
SPL {X  -162.820, Y  +555.861, Z    +0.000, E1   +42.349, E3 +375691.689}
SPL {X  -162.820, Y  +550.633, Z    +0.000, E1   +42.421, E3 +375703.219}
SPL {X  -162.820, Y  +546.534, Z    +0.000, E1   +42.268, E3 +375713.428}
SPL {X  -162.820, Y  +541.056, Z    +0.000, E1   +42.452, E3 +375724.944}
SPL {X  -162.820, Y  +535.223, Z    +0.000, E1   +42.386, E3 +375738.637}
SPL {X  -162.820, Y  +529.084, Z    +0.000, E1   +42.400, E3 +375752.560}
SPL {X  -162.820, Y  +524.911, Z    +0.000, E1   +42.325, E3 +375762.406}
SPL {X  -162.820, Y  +519.984, Z    +0.000, E1   +42.385, E3 +375773.477}
SPL {X  -162.820, Y  +514.684, Z    +0.000, E1   +42.289, E3 +375786.048}
SPL {X  -162.820, Y  +508.859, Z    +0.000, E1   +42.416, E3 +375798.699}
SPL {X  -162.820, Y  +501.651, Z    +0.000, E1   +42.423, E3 +375815.175}
SPL {X  -162.820, Y  +496.578, Z    +0.000, E1   +42.329, E3 +375827.084}
SPL {X  -162.820, Y  +493.739, Z    +0.000, E1   +42.260, E3 +375834.022}
SPL {X  -162.820, Y  +487.903, Z    +0.000, E1   +42.488, E3 +375846.108}
SPL {X  -162.820, Y  +484.250, Z    +0.000, E1   +42.201, E3 +375855.969}
SPL {X  -162.820, Y  +464.528, Z    +0.000, E1   +47.611, E3 +375864.792}
SPL {X  -162.820, Y  +459.899, Z    +0.000, E1   +47.097, E3 +375876.634}
SPL {X  -162.820, Y  +455.990, Z    +0.000, E1   +46.212, E3 +375889.708}
SPL {X  -162.820, Y  +452.032, Z    +0.000, E1   +45.224, E3 +375903.493}
SPL {X  -162.820, Y  +446.617, Z    +0.000, E1   +44.768, E3 +375917.580}
SPL {X  -162.820, Y  +437.902, Z    +0.000, E1   +44.900, E3 +375935.157}
SPL {X  -162.820, Y  +430.894, Z    +0.000, E1   +44.976, E3 +375949.142}
SPL {X  -162.820, Y  +425.053, Z    +0.000, E1   +44.824, E3 +375962.404}
SPL {X  -162.820, Y  +418.403, Z    +0.000, E1   +44.941, E3 +375975.518}
SPL {X  -162.820, Y  +412.479, Z    +0.000, E1   +44.780, E3 +375988.948}
SPL {X  -162.820, Y  +406.707, Z    +0.000, E1   +44.849, E3 +376000.521}
SPL {X  -162.820, Y  +400.166, Z    +0.000, E1   +44.948, E3 +376013.805}
SPL {X  -162.820, Y  +393.279, Z    +0.000, E1   +44.825, E3 +376028.808}
SPL {X  -162.820, Y  +387.883, Z    +0.000, E1   +44.837, E3 +376040.016}
SPL {X  -162.820, Y  +382.755, Z    +0.000, E1   +44.828, E3 +376050.809}
SPL {X  -162.796, Y  +377.700, Z    +0.000, E1   +44.829, E3 +376061.389}
SPL {X  -162.619, Y  +372.412, Z    +0.000, E1   +44.928, E3 +376071.849}
SPL {X  -162.170, Y  +365.961, Z    +0.000, E1   +44.802, E3 +376086.278}
SPL {X  -161.259, Y  +358.011, Z    +0.000, E1   +44.581, E3 +376104.205}
SPL {X  -160.417, Y  +352.631, Z    +0.000, E1   +44.411, E3 +376116.220}
SPL {X  -159.784, Y  +349.204, Z    +0.000, E1   +44.340, E3 +376123.812}
SPL {X  -158.853, Y  +344.776, Z    +0.000, E1   +44.148, E3 +376134.261}
SPL {X  -157.292, Y  +338.433, Z    +0.000, E1   +43.917, E3 +376148.940}
SPL {X  -155.654, Y  +332.729, Z    +0.000, E1   +43.534, E3 +376162.862}
SPL {X  -154.189, Y  +328.191, Z    +0.000, E1   +43.338, E3 +376173.358}
SPL {X  -149.333, Y  +315.614, Z    +0.000, E1   +46.650, E3 +376180.674}
SPL {X  -142.680, Y  +302.060, Z    +0.000, E1   +42.084, E3 +376247.018}
ENDSPLINE

SPLINE
SPL {X  -151.184, Y  +320.053, Z    +0.000, E1   +32.435, E3 +376314.261}
SPL {X  -158.917, Y  +345.064, Z    +0.000, E1   +21.858, E3 +376315.610}
SPL {X  -161.350, Y  +358.672, Z    +0.000, E1   +15.089, E3 +376318.312}
SPL {X  -162.491, Y  +370.147, Z    +0.000, E1    +8.815, E3 +376321.247}
SPL {X  -162.816, Y  +379.394, Z    +0.000, E1    +3.267, E3 +376321.075}
SPL {X  -162.820, Y  +384.427, Z    +0.000, E1    -0.390, E3 +376321.595}
SPL {X  -162.820, Y  +387.736, Z    +0.000, E1    -3.142, E3 +376320.875}
SPL {X  -162.820, Y  +391.456, Z    +0.000, E1    -6.603, E3 +376321.662}
SPL {X  -162.820, Y  +397.032, Z    +0.000, E1   -12.435, E3 +376321.109}
SPL {X  -162.820, Y  +406.111, Z    +0.000, E1   -22.010, E3 +376322.160}
SPL {X  -162.820, Y  +418.653, Z    +0.000, E1   -36.657, E3 +376316.513}
SPL {X  -162.820, Y  +440.590, Z    +0.000, E1   -50.152, E3 +376321.758}
SPL {X  -162.820, Y  +447.889, Z    +0.000, E1   -43.424, E3 +376352.904}
SPL {X  -162.820, Y  +478.087, Z    +0.000, E1   -45.903, E3 +376398.123}
ENDSPLINE

SPLINE
SPL {X  -162.820, Y  +474.900, Z    +0.000, E1   -42.394, E3 +376412.276}
ENDSPLINE

SPLINE
SPL {X  -162.820, Y  +480.895, Z    +0.000, E1   -42.223, E3 +376426.937}
SPL {X  -162.820, Y  +485.782, Z    +0.000, E1   -42.348, E3 +376437.283}
SPL {X  -162.820, Y  +489.480, Z    +0.000, E1   -42.230, E3 +376446.510}
SPL {X  -162.820, Y  +494.825, Z    +0.000, E1   -42.287, E3 +376458.457}
SPL {X  -162.820, Y  +501.023, Z    +0.000, E1   -42.347, E3 +376472.339}
SPL {X  -162.820, Y  +506.968, Z    +0.000, E1   -42.248, E3 +376486.530}
SPL {X  -162.820, Y  +513.215, Z    +0.000, E1   -42.304, E3 +376500.505}
SPL {X  -162.820, Y  +518.708, Z    +0.000, E1   -42.272, E3 +376513.226}
SPL {X  -162.820, Y  +525.147, Z    +0.000, E1   -42.298, E3 +376527.969}
SPL {X  -162.820, Y  +531.715, Z    +0.000, E1   -42.312, E3 +376542.794}
SPL {X  -162.820, Y  +537.459, Z    +0.000, E1   -42.308, E3 +376556.053}
SPL {X  -162.820, Y  +542.643, Z    +0.000, E1   -42.173, E3 +376568.646}
SPL {X  -162.820, Y  +547.830, Z    +0.000, E1   -42.372, E3 +376579.325}
SPL {X  -162.820, Y  +553.760, Z    +0.000, E1   -42.287, E3 +376593.601}
SPL {X  -162.820, Y  +561.114, Z    +0.000, E1   -42.336, E3 +376610.070}
SPL {X  -162.820, Y  +566.097, Z    +0.000, E1   -42.118, E3 +376622.680}
SPL {X  -162.820, Y  +571.654, Z    +0.000, E1   -42.313, E3 +376634.333}
SPL {X  -162.820, Y  +577.246, Z    +0.000, E1   -42.284, E3 +376647.299}
SPL {X  -162.820, Y  +582.233, Z    +0.000, E1   -42.188, E3 +376659.278}
SPL {X  -162.820, Y  +588.138, Z    +0.000, E1   -42.308, E3 +376672.176}
SPL {X  -162.820, Y  +593.999, Z    +0.000, E1   -42.301, E3 +376685.587}
SPL {X  -162.820, Y  +599.194, Z    +0.000, E1   -42.235, E3 +376697.891}
SPL {X  -162.820, Y  +604.595, Z    +0.000, E1   -42.290, E3 +376709.923}
SPL {X  -162.820, Y  +609.630, Z    +0.000, E1   -42.276, E3 +376721.549}
SPL {X  -162.820, Y  +614.392, Z    +0.000, E1   -42.242, E3 +376732.649}
SPL {X  -162.820, Y  +618.928, Z    +0.000, E1   -42.220, E3 +376743.174}
SPL {X  -162.820, Y  +625.176, Z    +0.000, E1   -42.323, E3 +376757.026}
SPL {X  -162.820, Y  +630.164, Z    +0.000, E1   -42.259, E3 +376768.636}
SPL {X  -162.820, Y  +635.892, Z    +0.000, E1   -42.319, E3 +376781.628}
SPL {X  -162.820, Y  +642.066, Z    +0.000, E1   -42.247, E3 +376796.036}
SPL {X  -162.820, Y  +646.907, Z    +0.000, E1   -42.249, E3 +376807.155}
SPL {X  -162.820, Y  +652.374, Z    +0.000, E1   -42.262, E3 +376819.593}
SPL {X  -162.820, Y  +657.439, Z    +0.000, E1   -42.251, E3 +376831.266}
SPL {X  -162.820, Y  +663.328, Z    +0.000, E1   -42.283, E3 +376844.668}
SPL {X  -162.820, Y  +669.078, Z    +0.000, E1   -42.263, E3 +376857.864}
SPL {X  -162.819, Y  +673.910, Z    +0.000, E1   -42.244, E3 +376869.059}
SPL {X  -162.729, Y  +678.944, Z    +0.000, E1   -42.273, E3 +376880.426}
SPL {X  -162.479, Y  +684.035, Z    +0.000, E1   -42.168, E3 +376892.764}
SPL {X  -162.026, Y  +689.560, Z    +0.000, E1   -42.192, E3 +376905.252}
SPL {X  -161.446, Y  +694.609, Z    +0.000, E1   -42.094, E3 +376917.384}
SPL {X  -160.681, Y  +699.806, Z    +0.000, E1   -41.866, E3 +376930.667}
SPL {X  -159.658, Y  +705.434, Z    +0.000, E1   -41.735, E3 +376944.297}
SPL {X  -158.502, Y  +710.748, Z    +0.000, E1   -41.532, E3 +376957.645}
SPL {X  -157.452, Y  +714.962, Z    +0.000, E1   -41.276, E3 +376968.640}
SPL {X  -156.530, Y  +718.319, Z    +0.000, E1   -41.164, E3 +376976.963}
SPL {X  -155.547, Y  +721.618, Z    +0.000, E1   -40.968, E3 +376985.587}
SPL {X  -151.388, Y  +733.433, Z    +0.000, E1   -44.269, E3 +376993.290}
SPL {X  -144.352, Y  +748.818, Z    +0.000, E1   -40.701, E3 +377062.324}
SPL {X  -143.859, Y  +749.757, Z    +0.000, E1   -39.148, E3 +377090.273}
ENDSPLINE

SPLINE
SPL {X  -159.245, Y  +707.432, Z    +0.000, E1   -21.244, E3 +377122.306}
SPL {X  -162.277, Y  +686.791, Z    +0.000, E1   -10.607, E3 +377123.716}
SPL {X  -162.766, Y  +677.687, Z    +0.000, E1    -5.239, E3 +377125.906}
SPL {X  -162.820, Y  +672.396, Z    +0.000, E1    -1.801, E3 +377126.695}
SPL {X  -162.820, Y  +667.851, Z    +0.000, E1    +1.551, E3 +377126.191}
SPL {X  -162.820, Y  +664.036, Z    +0.000, E1    +4.934, E3 +377126.910}
SPL {X  -162.820, Y  +661.024, Z    +0.000, E1    +7.880, E3 +377126.180}
SPL {X  -162.820, Y  +656.051, Z    +0.000, E1   +12.848, E3 +377127.047}
SPL {X  -162.820, Y  +650.794, Z    +0.000, E1   +18.580, E3 +377126.603}
SPL {X  -162.820, Y  +638.947, Z    +0.000, E1   +31.033, E3 +377124.951}
SPL {X  -162.820, Y  +608.150, Z    +0.000, E1   +43.921, E3 +377151.184}
SPL {X  -162.820, Y  +574.255, Z    +0.000, E1   +46.562, E3 +377200.978}
ENDSPLINE

SPLINE
SPL {X  -162.820, Y  +579.440, Z    +0.000, E1   +42.450, E3 +377214.165}
ENDSPLINE

SPLINE
SPL {X  -162.820, Y  +574.443, Z    +0.000, E1   +42.333, E3 +377226.260}
SPL {X  -162.820, Y  +568.554, Z    +0.000, E1   +42.362, E3 +377239.622}
SPL {X  -162.820, Y  +561.474, Z    +0.000, E1   +42.369, E3 +377255.808}
SPL {X  -162.820, Y  +555.861, Z    +0.000, E1   +42.349, E3 +377268.612}
SPL {X  -162.820, Y  +550.633, Z    +0.000, E1   +42.421, E3 +377280.142}
SPL {X  -162.820, Y  +546.534, Z    +0.000, E1   +42.268, E3 +377290.352}
SPL {X  -162.820, Y  +539.632, Z    +0.000, E1   +42.488, E3 +377305.073}
SPL {X  -162.820, Y  +533.959, Z    +0.000, E1   +42.310, E3 +377318.770}
SPL {X  -162.820, Y  +527.661, Z    +0.000, E1   +42.425, E3 +377332.765}
SPL {X  -162.820, Y  +521.246, Z    +0.000, E1   +42.365, E3 +377347.518}
SPL {X  -162.820, Y  +515.708, Z    +0.000, E1   +42.333, E3 +377360.481}
SPL {X  -162.820, Y  +510.265, Z    +0.000, E1   +42.390, E3 +377372.442}
SPL {X  -162.820, Y  +505.746, Z    +0.000, E1   +42.400, E3 +377382.755}
SPL {X  -162.820, Y  +500.461, Z    +0.000, E1   +42.387, E3 +377394.882}
SPL {X  -162.820, Y  +494.841, Z    +0.000, E1   +42.316, E3 +377408.208}
SPL {X  -162.820, Y  +486.958, Z    +0.000, E1   +42.460, E3 +377425.501}
SPL {X  -162.820, Y  +464.528, Z    +0.000, E1   +47.611, E3 +377441.715}
SPL {X  -162.820, Y  +458.830, Z    +0.000, E1   +46.994, E3 +377456.393}
SPL {X  -162.820, Y  +455.537, Z    +0.000, E1   +45.900, E3 +377469.212}
SPL {X  -162.820, Y  +452.032, Z    +0.000, E1   +45.224, E3 +377480.416}
SPL {X  -162.820, Y  +446.617, Z    +0.000, E1   +44.768, E3 +377494.503}
SPL {X  -162.820, Y  +440.464, Z    +0.000, E1   +44.845, E3 +377506.805}
SPL {X  -162.820, Y  +435.902, Z    +0.000, E1   +44.853, E3 +377516.328}
SPL {X  -162.820, Y  +429.336, Z    +0.000, E1   +44.917, E3 +377529.847}
SPL {X  -162.820, Y  +423.193, Z    +0.000, E1   +44.819, E3 +377543.106}
SPL {X  -162.820, Y  +416.810, Z    +0.000, E1   +44.932, E3 +377555.994}
SPL {X  -162.820, Y  +408.782, Z    +0.000, E1   +44.820, E3 +377573.424}
SPL {X  -162.820, Y  +401.619, Z    +0.000, E1   +44.978, E3 +377587.346}
SPL {X  -162.820, Y  +394.771, Z    +0.000, E1   +44.856, E3 +377602.585}
SPL {X  -162.820, Y  +387.883, Z    +0.000, E1   +44.837, E3 +377616.939}
SPL {X  -162.820, Y  +382.755, Z    +0.000, E1   +44.828, E3 +377627.732}
SPL {X  -162.796, Y  +377.700, Z    +0.000, E1   +44.829, E3 +377638.312}
SPL {X  -162.619, Y  +372.412, Z    +0.000, E1   +44.928, E3 +377648.772}
SPL {X  -162.311, Y  +367.633, Z    +0.000, E1   +44.798, E3 +377659.539}
SPL {X  -161.766, Y  +362.002, Z    +0.000, E1   +44.644, E3 +377672.297}
SPL {X  -161.043, Y  +356.508, Z    +0.000, E1   +44.528, E3 +377684.412}
SPL {X  -160.070, Y  +350.699, Z    +0.000, E1   +44.409, E3 +377697.364}
SPL {X  -158.853, Y  +344.776, Z    +0.000, E1   +44.148, E3 +377711.184}
SPL {X  -157.292, Y  +338.433, Z    +0.000, E1   +43.917, E3 +377725.863}
SPL {X  -155.654, Y  +332.729, Z    +0.000, E1   +43.534, E3 +377739.785}
SPL {X  -154.189, Y  +328.191, Z    +0.000, E1   +43.338, E3 +377750.281}
SPL {X  -149.333, Y  +315.614, Z    +0.000, E1   +46.650, E3 +377757.597}
SPL {X  -142.680, Y  +302.060, Z    +0.000, E1   +42.084, E3 +377823.941}
ENDSPLINE

SPLINE
SPL {X  -151.184, Y  +320.053, Z    +0.000, E1   +32.435, E3 +377891.184}
SPL {X  -158.917, Y  +345.064, Z    +0.000, E1   +21.858, E3 +377892.533}
SPL {X  -161.350, Y  +358.672, Z    +0.000, E1   +15.089, E3 +377895.235}
SPL {X  -162.491, Y  +370.147, Z    +0.000, E1    +8.815, E3 +377898.170}
SPL {X  -162.816, Y  +379.394, Z    +0.000, E1    +3.267, E3 +377897.998}
SPL {X  -162.820, Y  +384.427, Z    +0.000, E1    -0.390, E3 +377898.518}
SPL {X  -162.820, Y  +387.736, Z    +0.000, E1    -3.142, E3 +377897.798}
SPL {X  -162.820, Y  +391.456, Z    +0.000, E1    -6.603, E3 +377898.585}
SPL {X  -162.820, Y  +397.032, Z    +0.000, E1   -12.435, E3 +377898.032}
SPL {X  -162.820, Y  +406.111, Z    +0.000, E1   -22.010, E3 +377899.083}
SPL {X  -162.820, Y  +418.653, Z    +0.000, E1   -36.657, E3 +377893.436}
SPL {X  -162.820, Y  +440.590, Z    +0.000, E1   -50.152, E3 +377898.681}
SPL {X  -162.820, Y  +447.889, Z    +0.000, E1   -43.424, E3 +377929.827}
SPL {X  -162.820, Y  +478.087, Z    +0.000, E1   -45.903, E3 +377975.046}
ENDSPLINE

SPLINE
SPL {X  -162.820, Y  +472.818, Z    +0.000, E1   -42.437, E3 +377983.987}
ENDSPLINE

SPLINE
SPL {X  -162.820, Y  +476.137, Z    +0.000, E1   -42.304, E3 +377992.401}
SPL {X  -162.820, Y  +480.895, Z    +0.000, E1   -42.223, E3 +378003.860}
SPL {X  -162.820, Y  +488.112, Z    +0.000, E1   -42.323, E3 +378019.941}
SPL {X  -162.820, Y  +496.300, Z    +0.000, E1   -42.332, E3 +378038.654}
SPL {X  -162.820, Y  +503.162, Z    +0.000, E1   -42.272, E3 +378054.571}
SPL {X  -162.820, Y  +508.157, Z    +0.000, E1   -42.280, E3 +378065.897}
SPL {X  -162.820, Y  +513.215, Z    +0.000, E1   -42.304, E3 +378077.428}
SPL {X  -162.820, Y  +520.311, Z    +0.000, E1   -42.317, E3 +378093.726}
SPL {X  -162.820, Y  +526.529, Z    +0.000, E1   -42.247, E3 +378108.195}
SPL {X  -162.820, Y  +532.723, Z    +0.000, E1   -42.344, E3 +378121.937}
SPL {X  -162.820, Y  +538.500, Z    +0.000, E1   -42.256, E3 +378135.558}
SPL {X  -162.820, Y  +542.643, Z    +0.000, E1   -42.173, E3 +378145.569}
SPL {X  -162.820, Y  +549.160, Z    +0.000, E1   -42.387, E3 +378159.327}
SPL {X  -162.820, Y  +554.884, Z    +0.000, E1   -42.207, E3 +378173.413}
SPL {X  -162.820, Y  +559.897, Z    +0.000, E1   -42.319, E3 +378184.198}
SPL {X  -162.820, Y  +565.154, Z    +0.000, E1   -42.205, E3 +378197.044}
SPL {X  -162.820, Y  +571.654, Z    +0.000, E1   -42.313, E3 +378211.256}
SPL {X  -162.820, Y  +577.246, Z    +0.000, E1   -42.284, E3 +378224.222}
SPL {X  -162.820, Y  +582.233, Z    +0.000, E1   -42.188, E3 +378236.201}
SPL {X  -162.820, Y  +588.138, Z    +0.000, E1   -42.308, E3 +378249.100}
SPL {X  -162.820, Y  +593.999, Z    +0.000, E1   -42.301, E3 +378262.510}
SPL {X  -162.820, Y  +599.194, Z    +0.000, E1   -42.235, E3 +378274.814}
SPL {X  -162.820, Y  +604.595, Z    +0.000, E1   -42.290, E3 +378286.846}
SPL {X  -162.820, Y  +609.630, Z    +0.000, E1   -42.276, E3 +378298.472}
SPL {X  -162.820, Y  +614.392, Z    +0.000, E1   -42.242, E3 +378309.572}
SPL {X  -162.820, Y  +620.424, Z    +0.000, E1   -42.277, E3 +378323.319}
SPL {X  -162.820, Y  +626.430, Z    +0.000, E1   -42.291, E3 +378336.869}
SPL {X  -162.820, Y  +631.865, Z    +0.000, E1   -42.327, E3 +378349.163}
SPL {X  -162.820, Y  +637.189, Z    +0.000, E1   -42.236, E3 +378361.837}
SPL {X  -162.820, Y  +642.066, Z    +0.000, E1   -42.247, E3 +378372.959}
SPL {X  -162.820, Y  +646.907, Z    +0.000, E1   -42.249, E3 +378384.078}
SPL {X  -162.820, Y  +652.374, Z    +0.000, E1   -42.262, E3 +378396.516}
SPL {X  -162.820, Y  +658.634, Z    +0.000, E1   -42.281, E3 +378410.873}
SPL {X  -162.820, Y  +664.480, Z    +0.000, E1   -42.257, E3 +378424.268}
SPL {X  -162.820, Y  +669.078, Z    +0.000, E1   -42.263, E3 +378434.788}
SPL {X  -162.819, Y  +673.910, Z    +0.000, E1   -42.244, E3 +378445.982}
SPL {X  -162.729, Y  +678.944, Z    +0.000, E1   -42.273, E3 +378457.349}
SPL {X  -162.479, Y  +684.035, Z    +0.000, E1   -42.168, E3 +378469.687}
SPL {X  -162.026, Y  +689.560, Z    +0.000, E1   -42.192, E3 +378482.175}
SPL {X  -161.446, Y  +694.609, Z    +0.000, E1   -42.094, E3 +378494.307}
SPL {X  -160.889, Y  +698.503, Z    +0.000, E1   -41.849, E3 +378504.581}
SPL {X  -160.100, Y  +703.138, Z    +0.000, E1   -41.824, E3 +378515.440}
SPL {X  -159.403, Y  +706.682, Z    +0.000, E1   -41.618, E3 +378524.618}
SPL {X  -158.502, Y  +710.748, Z    +0.000, E1   -41.532, E3 +378534.568}
SPL {X  -157.452, Y  +714.962, Z    +0.000, E1   -41.276, E3 +378545.563}
SPL {X  -156.258, Y  +719.258, Z    +0.000, E1   -41.133, E3 +378556.308}
SPL {X  -155.356, Y  +722.233, Z    +0.000, E1   -40.927, E3 +378564.097}
SPL {X  -151.388, Y  +733.433, Z    +0.000, E1   -44.269, E3 +378570.213}
SPL {X  -144.352, Y  +748.818, Z    +0.000, E1   -40.701, E3 +378639.247}
SPL {X  -143.859, Y  +749.757, Z    +0.000, E1   -39.148, E3 +378667.196}
ENDSPLINE

SPLINE
SPL {X  -159.245, Y  +707.432, Z    +0.000, E1   -21.244, E3 +378699.229}
SPL {X  -162.277, Y  +686.791, Z    +0.000, E1   -10.607, E3 +378700.639}
SPL {X  -162.766, Y  +677.687, Z    +0.000, E1    -5.239, E3 +378702.829}
SPL {X  -162.820, Y  +671.059, Z    +0.000, E1    -0.934, E3 +378703.185}
SPL {X  -162.820, Y  +666.960, Z    +0.000, E1    +2.343, E3 +378703.462}
SPL {X  -162.820, Y  +662.610, Z    +0.000, E1    +6.209, E3 +378703.488}
SPL {X  -162.820, Y  +654.280, Z    +0.000, E1   +14.617, E3 +378703.821}
SPL {X  -162.820, Y  +638.947, Z    +0.000, E1   +31.033, E3 +378701.874}
SPL {X  -162.820, Y  +608.150, Z    +0.000, E1   +43.921, E3 +378728.107}
SPL {X  -162.820, Y  +574.255, Z    +0.000, E1   +46.562, E3 +378777.901}
ENDSPLINE

SPLINE
SPL {X  -162.820, Y  +579.440, Z    +0.000, E1   +42.450, E3 +378791.088}
ENDSPLINE

SPLINE
SPL {X  -162.820, Y  +574.443, Z    +0.000, E1   +42.333, E3 +378803.183}
SPL {X  -162.820, Y  +568.554, Z    +0.000, E1   +42.362, E3 +378816.545}
SPL {X  -162.820, Y  +563.699, Z    +0.000, E1   +42.375, E3 +378827.402}
SPL {X  -162.820, Y  +560.278, Z    +0.000, E1   +42.308, E3 +378835.687}
SPL {X  -162.820, Y  +554.421, Z    +0.000, E1   +42.414, E3 +378848.555}
SPL {X  -162.820, Y  +547.774, Z    +0.000, E1   +42.344, E3 +378864.128}
SPL {X  -162.820, Y  +541.056, Z    +0.000, E1   +42.452, E3 +378878.790}
SPL {X  -162.820, Y  +535.223, Z    +0.000, E1   +42.386, E3 +378892.484}
SPL {X  -162.820, Y  +529.084, Z    +0.000, E1   +42.400, E3 +378906.406}
SPL {X  -162.820, Y  +522.568, Z    +0.000, E1   +42.385, E3 +378921.436}
SPL {X  -162.820, Y  +515.708, Z    +0.000, E1   +42.333, E3 +378937.404}
SPL {X  -162.820, Y  +508.859, Z    +0.000, E1   +42.416, E3 +378952.546}
SPL {X  -162.820, Y  +501.651, Z    +0.000, E1   +42.423, E3 +378969.021}
SPL {X  -162.820, Y  +494.841, Z    +0.000, E1   +42.316, E3 +378985.131}
SPL {X  -162.820, Y  +487.903, Z    +0.000, E1   +42.488, E3 +378999.954}
SPL {X  -162.820, Y  +484.250, Z    +0.000, E1   +42.201, E3 +379009.815}
SPL {X  -162.820, Y  +466.305, Z    +0.000, E1   +47.564, E3 +379015.432}
SPL {X  -162.820, Y  +460.790, Z    +0.000, E1   +47.323, E3 +379027.607}
SPL {X  -162.820, Y  +455.990, Z    +0.000, E1   +46.212, E3 +379043.554}
SPL {X  -162.820, Y  +452.032, Z    +0.000, E1   +45.224, E3 +379057.340}
ENDSPLINE

SPLINE
SPL {X  -162.820, Y  +466.981, Z    +0.000, E1   +37.285, E3 +379069.268}
ENDSPLINE

SPLINE
SPL {X  -162.820, Y  +462.598, Z    +0.000, E1   +37.325, E3 +379080.999}
SPL {X  -162.820, Y  +459.177, Z    +0.000, E1   +37.207, E3 +379091.026}
SPL {X  -162.820, Y  +453.939, Z    +0.000, E1   +37.397, E3 +379104.379}
SPL {X  -162.820, Y  +448.311, Z    +0.000, E1   +37.333, E3 +379120.040}
SPL {X  -162.820, Y  +443.351, Z    +0.000, E1   +37.335, E3 +379133.569}
SPL {X  -162.820, Y  +438.727, Z    +0.000, E1   +37.289, E3 +379146.442}
SPL {X  -162.820, Y  +434.320, Z    +0.000, E1   +37.343, E3 +379158.152}
SPL {X  -162.820, Y  +430.091, Z    +0.000, E1   +37.424, E3 +379169.152}
SPL {X  -162.820, Y  +426.177, Z    +0.000, E1   +37.250, E3 +379180.974}
SPL {X  -162.820, Y  +420.241, Z    +0.000, E1   +37.355, E3 +379196.681}
SPL {X  -162.820, Y  +415.595, Z    +0.000, E1   +37.375, E3 +379209.021}
SPL {X  -162.820, Y  +411.860, Z    +0.000, E1   +37.402, E3 +379219.124}
SPL {X  -162.820, Y  +407.726, Z    +0.000, E1   +37.291, E3 +379231.072}
SPL {X  -162.820, Y  +403.543, Z    +0.000, E1   +37.305, E3 +379242.417}
SPL {X  -162.820, Y  +399.300, Z    +0.000, E1   +37.355, E3 +379253.701}
SPL {X  -162.820, Y  +395.182, Z    +0.000, E1   +37.347, E3 +379264.991}
SPL {X  -162.820, Y  +390.797, Z    +0.000, E1   +37.358, E3 +379276.903}
SPL {X  -162.820, Y  +386.671, Z    +0.000, E1   +37.363, E3 +379288.084}
SPL {X  -162.820, Y  +382.174, Z    +0.000, E1   +37.329, E3 +379300.661}
SPL {X  -162.785, Y  +377.133, Z    +0.000, E1   +37.299, E3 +379314.590}
SPL {X  -162.623, Y  +372.484, Z    +0.000, E1   +37.337, E3 +379327.030}
SPL {X  -162.331, Y  +367.894, Z    +0.000, E1   +37.251, E3 +379340.143}
SPL {X  -161.920, Y  +363.407, Z    +0.000, E1   +37.164, E3 +379352.877}
SPL {X  -161.482, Y  +359.669, Z    +0.000, E1   +37.064, E3 +379363.661}
SPL {X  -160.943, Y  +355.851, Z    +0.000, E1   +37.136, E3 +379373.648}
SPL {X  -160.493, Y  +353.069, Z    +0.000, E1   +36.789, E3 +379383.300}
SPL {X  -159.837, Y  +349.474, Z    +0.000, E1   +36.824, E3 +379392.966}
SPL {X  -159.171, Y  +346.224, Z    +0.000, E1   +36.747, E3 +379402.242}
SPL {X  -158.248, Y  +342.188, Z    +0.000, E1   +36.583, E3 +379414.405}
SPL {X  -153.520, Y  +326.260, Z    +0.000, E1   +41.363, E3 +379427.057}
SPL {X  -150.942, Y  +319.452, Z    +0.000, E1   +36.529, E3 +379483.414}
ENDSPLINE

SPLINE
SPL {X  -159.264, Y  +346.659, Z    +0.000, E1   +22.083, E3 +379523.988}
SPL {X  -161.245, Y  +357.907, Z    +0.000, E1   +16.095, E3 +379537.421}
SPL {X  -162.746, Y  +375.590, Z    +0.000, E1    +6.280, E3 +379537.010}
SPL {X  -162.820, Y  +384.478, Z    +0.000, E1    +0.434, E3 +379537.679}
SPL {X  -162.820, Y  +389.965, Z    +0.000, E1    -3.918, E3 +379537.390}
SPL {X  -162.820, Y  +394.532, Z    +0.000, E1    -7.849, E3 +379538.939}
SPL {X  -162.820, Y  +400.765, Z    +0.000, E1   -14.108, E3 +379536.405}
SPL {X  -162.820, Y  +411.829, Z    +0.000, E1   -24.195, E3 +379538.483}
SPL {X  -162.820, Y  +434.900, Z    +0.000, E1   -34.666, E3 +379565.848}
SPL {X  -162.820, Y  +465.031, Z    +0.000, E1   -41.710, E3 +379603.520}
SPL {X  -162.820, Y  +465.893, Z    +0.000, E1   -40.572, E3 +379612.049}
ENDSPLINE

SPLINE
SPL {X  -162.820, Y  +458.794, Z    +0.000, E1   -36.100, E3 +379620.778}
ENDSPLINE

SPLINE
SPL {X  -162.820, Y  +461.779, Z    +0.000, E1   -35.988, E3 +379629.974}
SPL {X  -162.820, Y  +465.690, Z    +0.000, E1   -36.140, E3 +379640.269}
SPL {X  -162.820, Y  +470.432, Z    +0.000, E1   -36.100, E3 +379654.152}
SPL {X  -162.820, Y  +475.701, Z    +0.000, E1   -36.157, E3 +379668.779}
SPL {X  -162.820, Y  +479.954, Z    +0.000, E1   -36.086, E3 +379681.319}
SPL {X  -162.820, Y  +485.438, Z    +0.000, E1   -36.112, E3 +379697.037}
SPL {X  -162.820, Y  +490.843, Z    +0.000, E1   -36.087, E3 +379712.450}
SPL {X  -162.820, Y  +494.712, Z    +0.000, E1   -36.164, E3 +379722.963}
SPL {X  -162.820, Y  +497.796, Z    +0.000, E1   -36.022, E3 +379732.669}
SPL {X  -162.820, Y  +502.146, Z    +0.000, E1   -36.123, E3 +379744.538}
SPL {X  -162.820, Y  +505.688, Z    +0.000, E1   -36.050, E3 +379755.020}
SPL {X  -162.820, Y  +509.364, Z    +0.000, E1   -36.084, E3 +379765.391}
SPL {X  -162.820, Y  +515.001, Z    +0.000, E1   -36.183, E3 +379781.029}
SPL {X  -162.820, Y  +520.482, Z    +0.000, E1   -36.096, E3 +379797.074}
SPL {X  -162.820, Y  +525.226, Z    +0.000, E1   -36.081, E3 +379810.742}
SPL {X  -162.820, Y  +530.908, Z    +0.000, E1   -36.155, E3 +379826.599}
SPL {X  -162.820, Y  +536.031, Z    +0.000, E1   -36.058, E3 +379841.718}
SPL {X  -162.820, Y  +541.179, Z    +0.000, E1   -36.085, E3 +379856.359}
SPL {X  -162.820, Y  +546.355, Z    +0.000, E1   -36.114, E3 +379870.903}
SPL {X  -162.820, Y  +551.776, Z    +0.000, E1   -36.108, E3 +379886.537}
SPL {X  -162.820, Y  +556.944, Z    +0.000, E1   -36.118, E3 +379901.108}
SPL {X  -162.820, Y  +561.684, Z    +0.000, E1   -36.118, E3 +379914.700}
SPL {X  -162.820, Y  +566.500, Z    +0.000, E1   -36.073, E3 +379928.702}
SPL {X  -162.820, Y  +571.734, Z    +0.000, E1   -36.094, E3 +379943.632}
SPL {X  -162.820, Y  +576.887, Z    +0.000, E1   -36.084, E3 +379958.325}
SPL {X  -162.820, Y  +581.763, Z    +0.000, E1   -36.093, E3 +379972.262}
SPL {X  -162.820, Y  +586.693, Z    +0.000, E1   -36.086, E3 +379986.367}
SPL {X  -162.820, Y  +591.665, Z    +0.000, E1   -36.045, E3 +380000.895}
SPL {X  -162.820, Y  +596.059, Z    +0.000, E1   -36.124, E3 +380012.827}
SPL {X  -162.820, Y  +598.788, Z    +0.000, E1   -36.102, E3 +380020.738}
SPL {X  -162.820, Y  +602.243, Z    +0.000, E1   -36.085, E3 +380030.804}
SPL {X  -162.820, Y  +605.848, Z    +0.000, E1   -36.070, E3 +380041.125}
SPL {X  -162.820, Y  +609.375, Z    +0.000, E1   -36.084, E3 +380051.176}
SPL {X  -162.820, Y  +612.959, Z    +0.000, E1   -36.034, E3 +380061.696}
SPL {X  -162.820, Y  +616.897, Z    +0.000, E1   -36.061, E3 +380072.844}
SPL {X  -162.820, Y  +621.516, Z    +0.000, E1   -36.072, E3 +380086.043}
SPL {X  -162.820, Y  +626.243, Z    +0.000, E1   -36.105, E3 +380099.286}
SPL {X  -162.820, Y  +630.571, Z    +0.000, E1   -36.057, E3 +380111.987}
SPL {X  -162.820, Y  +635.505, Z    +0.000, E1   -36.079, E3 +380125.993}
SPL {X  -162.820, Y  +641.277, Z    +0.000, E1   -36.126, E3 +380142.286}
SPL {X  -162.820, Y  +646.320, Z    +0.000, E1   -36.078, E3 +380156.851}
SPL {X  -162.820, Y  +651.289, Z    +0.000, E1   -36.059, E3 +380171.307}
SPL {X  -162.820, Y  +656.677, Z    +0.000, E1   -36.110, E3 +380186.321}
SPL {X  -162.820, Y  +661.560, Z    +0.000, E1   -36.068, E3 +380200.584}
SPL {X  -162.820, Y  +666.386, Z    +0.000, E1   -36.048, E3 +380214.468}
SPL {X  -162.820, Y  +671.104, Z    +0.000, E1   -36.061, E3 +380227.887}
SPL {X  -162.787, Y  +676.764, Z    +0.000, E1   -36.126, E3 +380243.787}
SPL {X  -162.633, Y  +681.311, Z    +0.000, E1   -35.984, E3 +380257.475}
SPL {X  -162.367, Y  +685.641, Z    +0.000, E1   -36.000, E3 +380269.883}
SPL {X  -161.948, Y  +690.331, Z    +0.000, E1   -35.960, E3 +380283.479}
SPL {X  -161.544, Y  +693.846, Z    +0.000, E1   -35.908, E3 +380293.754}
SPL {X  -161.078, Y  +697.256, Z    +0.000, E1   -35.797, E3 +380304.260}
SPL {X  -160.313, Y  +701.964, Z    +0.000, E1   -35.709, E3 +380318.335}
SPL {X  -159.622, Y  +705.613, Z    +0.000, E1   -35.430, E3 +380330.275}
SPL {X  -158.758, Y  +709.640, Z    +0.000, E1   -35.380, E3 +380342.282}
SPL {X  -155.037, Y  +723.239, Z    +0.000, E1   -39.382, E3 +380355.167}
SPL {X  -152.141, Y  +731.494, Z    +0.000, E1   -35.181, E3 +380413.973}
ENDSPLINE

SPLINE
SPL {X  -160.133, Y  +702.956, Z    +0.000, E1   -19.806, E3 +380457.511}
SPL {X  -161.979, Y  +690.023, Z    +0.000, E1   -12.991, E3 +380460.427}
SPL {X  -162.641, Y  +681.139, Z    +0.000, E1    -7.893, E3 +380462.519}
SPL {X  -162.820, Y  +673.062, Z    +0.000, E1    -2.992, E3 +380461.486}
SPL {X  -162.820, Y  +665.516, Z    +0.000, E1    +2.410, E3 +380463.326}
SPL {X  -162.820, Y  +657.781, Z    +0.000, E1    +9.391, E3 +380460.990}
SPL {X  -162.820, Y  +648.706, Z    +0.000, E1   +17.761, E3 +380462.742}
SPL {X  -162.820, Y  +629.267, Z    +0.000, E1   +31.872, E3 +380472.947}
SPL {X  -162.820, Y  +620.680, Z    +0.000, E1   +34.107, E3 +380486.997}
SPL {X  -162.820, Y  +601.185, Z    +0.000, E1   +39.430, E3 +380510.504}
SPL {X  -162.820, Y  +599.927, Z    +0.000, E1   +35.241, E3 +380537.083}
SPL {X  -162.820, Y  +599.021, Z    +0.000, E1   +33.912, E3 +380548.133}
SPL {X  -162.820, Y  +595.170, Z    +0.000, E1   +33.784, E3 +380561.039}
SPL {X  -162.820, Y  +589.785, Z    +0.000, E1   +33.904, E3 +380577.036}
SPL {X  -162.820, Y  +584.646, Z    +0.000, E1   +33.882, E3 +380593.105}
SPL {X  -162.820, Y  +579.919, Z    +0.000, E1   +33.857, E3 +380607.893}
SPL {X  -162.820, Y  +574.615, Z    +0.000, E1   +33.920, E3 +380624.067}
SPL {X  -162.820, Y  +569.298, Z    +0.000, E1   +33.851, E3 +380640.929}
SPL {X  -162.820, Y  +563.983, Z    +0.000, E1   +33.916, E3 +380657.070}
SPL {X  -162.820, Y  +559.395, Z    +0.000, E1   +33.796, E3 +380671.951}
SPL {X  -162.820, Y  +554.453, Z    +0.000, E1   +33.841, E3 +380687.176}
SPL {X  -162.820, Y  +549.726, Z    +0.000, E1   +33.905, E3 +380701.279}
SPL {X  -162.820, Y  +545.760, Z    +0.000, E1   +33.901, E3 +380713.675}
SPL {X  -162.820, Y  +541.668, Z    +0.000, E1   +33.787, E3 +380727.075}
SPL {X  -162.820, Y  +537.061, Z    +0.000, E1   +33.897, E3 +380740.734}
SPL {X  -162.820, Y  +532.164, Z    +0.000, E1   +33.861, E3 +380756.207}
SPL {X  -162.820, Y  +526.783, Z    +0.000, E1   +33.870, E3 +380772.890}
SPL {X  -162.820, Y  +521.520, Z    +0.000, E1   +33.826, E3 +380789.537}
SPL {X  -162.820, Y  +516.814, Z    +0.000, E1   +33.917, E3 +380803.438}
SPL {X  -162.820, Y  +512.685, Z    +0.000, E1   +33.830, E3 +380816.881}
SPL {X  -162.820, Y  +508.888, Z    +0.000, E1   +33.871, E3 +380828.296}
SPL {X  -162.820, Y  +505.651, Z    +0.000, E1   +33.839, E3 +380838.613}
SPL {X  -162.820, Y  +500.931, Z    +0.000, E1   +34.256, E3 +380850.487}
SPL {X  -162.820, Y  +481.122, Z    +0.000, E1   +41.279, E3 +380860.751}
SPL {X  -162.820, Y  +478.698, Z    +0.000, E1   +40.526, E3 +380871.100}
SPL {X  -162.820, Y  +475.203, Z    +0.000, E1   +39.596, E3 +380885.559}
SPL {X  -162.820, Y  +472.097, Z    +0.000, E1   +38.411, E3 +380900.526}
SPL {X  -162.820, Y  +469.308, Z    +0.000, E1   +37.839, E3 +380911.330}
SPL {X  -162.820, Y  +467.216, Z    +0.000, E1   +37.215, E3 +380920.897}
SPL {X  -162.820, Y  +462.598, Z    +0.000, E1   +37.325, E3 +380932.851}
SPL {X  -162.820, Y  +457.832, Z    +0.000, E1   +37.294, E3 +380946.138}
SPL {X  -162.820, Y  +452.986, Z    +0.000, E1   +37.368, E3 +380958.871}
SPL {X  -162.820, Y  +447.084, Z    +0.000, E1   +37.389, E3 +380975.062}
SPL {X  -162.820, Y  +440.036, Z    +0.000, E1   +37.326, E3 +380994.680}
SPL {X  -162.820, Y  +434.320, Z    +0.000, E1   +37.343, E3 +381010.003}
SPL {X  -162.820, Y  +430.091, Z    +0.000, E1   +37.424, E3 +381021.003}
SPL {X  -162.820, Y  +426.177, Z    +0.000, E1   +37.250, E3 +381032.826}
SPL {X  -162.820, Y  +421.391, Z    +0.000, E1   +37.346, E3 +381045.290}
SPL {X  -162.820, Y  +416.811, Z    +0.000, E1   +37.348, E3 +381057.824}
SPL {X  -162.820, Y  +411.860, Z    +0.000, E1   +37.402, E3 +381070.976}
SPL {X  -162.820, Y  +407.726, Z    +0.000, E1   +37.291, E3 +381082.924}
SPL {X  -162.820, Y  +403.543, Z    +0.000, E1   +37.305, E3 +381094.269}
SPL {X  -162.820, Y  +399.300, Z    +0.000, E1   +37.355, E3 +381105.553}
SPL {X  -162.820, Y  +395.182, Z    +0.000, E1   +37.347, E3 +381116.842}
SPL {X  -162.820, Y  +390.797, Z    +0.000, E1   +37.358, E3 +381128.755}
SPL {X  -162.820, Y  +386.671, Z    +0.000, E1   +37.363, E3 +381139.936}
SPL {X  -162.820, Y  +382.174, Z    +0.000, E1   +37.329, E3 +381152.513}
SPL {X  -162.785, Y  +377.133, Z    +0.000, E1   +37.299, E3 +381166.442}
SPL {X  -162.576, Y  +371.586, Z    +0.000, E1   +37.322, E3 +381181.555}
SPL {X  -162.256, Y  +366.963, Z    +0.000, E1   +37.251, E3 +381194.444}
SPL {X  -161.920, Y  +363.407, Z    +0.000, E1   +37.164, E3 +381204.729}
SPL {X  -161.482, Y  +359.669, Z    +0.000, E1   +37.064, E3 +381215.513}
SPL {X  -160.943, Y  +355.851, Z    +0.000, E1   +37.136, E3 +381225.500}
SPL {X  -160.493, Y  +353.069, Z    +0.000, E1   +36.789, E3 +381235.152}
SPL {X  -159.837, Y  +349.474, Z    +0.000, E1   +36.824, E3 +381244.817}
SPL {X  -158.862, Y  +344.820, Z    +0.000, E1   +36.732, E3 +381258.180}
SPL {X  -157.959, Y  +341.011, Z    +0.000, E1   +36.448, E3 +381270.077}
SPL {X  -153.520, Y  +326.260, Z    +0.000, E1   +41.363, E3 +381278.909}
SPL {X  -150.942, Y  +319.452, Z    +0.000, E1   +36.529, E3 +381335.266}
ENDSPLINE

SPLINE
SPL {X  -159.264, Y  +346.659, Z    +0.000, E1   +22.083, E3 +381375.840}
SPL {X  -161.245, Y  +357.907, Z    +0.000, E1   +16.095, E3 +381389.273}
SPL {X  -162.697, Y  +374.161, Z    +0.000, E1    +7.119, E3 +381387.262}
SPL {X  -162.820, Y  +380.878, Z    +0.000, E1    +2.854, E3 +381390.094}
SPL {X  -162.820, Y  +385.313, Z    +0.000, E1    -0.228, E3 +381389.874}
SPL {X  -162.820, Y  +389.965, Z    +0.000, E1    -3.918, E3 +381389.242}
SPL {X  -162.820, Y  +394.532, Z    +0.000, E1    -7.849, E3 +381390.791}
SPL {X  -162.820, Y  +400.765, Z    +0.000, E1   -14.108, E3 +381388.257}
SPL {X  -162.820, Y  +411.829, Z    +0.000, E1   -24.195, E3 +381390.335}
SPL {X  -162.820, Y  +434.900, Z    +0.000, E1   -34.666, E3 +381417.699}
SPL {X  -162.820, Y  +465.440, Z    +0.000, E1   -41.264, E3 +381459.007}
ENDSPLINE

SPLINE
SPL {X  -162.820, Y  +458.794, Z    +0.000, E1   -36.100, E3 +381472.630}
ENDSPLINE

SPLINE
SPL {X  -162.820, Y  +461.779, Z    +0.000, E1   -35.988, E3 +381481.826}
SPL {X  -162.820, Y  +467.031, Z    +0.000, E1   -36.178, E3 +381495.897}
SPL {X  -162.820, Y  +471.524, Z    +0.000, E1   -36.022, E3 +381509.450}
SPL {X  -162.820, Y  +475.701, Z    +0.000, E1   -36.157, E3 +381520.631}
SPL {X  -162.820, Y  +479.954, Z    +0.000, E1   -36.086, E3 +381533.171}
SPL {X  -162.820, Y  +485.438, Z    +0.000, E1   -36.112, E3 +381548.889}
SPL {X  -162.820, Y  +490.843, Z    +0.000, E1   -36.087, E3 +381564.302}
SPL {X  -162.820, Y  +494.712, Z    +0.000, E1   -36.164, E3 +381574.815}
SPL {X  -162.820, Y  +497.796, Z    +0.000, E1   -36.022, E3 +381584.521}
SPL {X  -162.820, Y  +502.146, Z    +0.000, E1   -36.123, E3 +381596.390}
SPL {X  -162.820, Y  +505.688, Z    +0.000, E1   -36.050, E3 +381606.872}
SPL {X  -162.820, Y  +509.364, Z    +0.000, E1   -36.084, E3 +381617.243}
SPL {X  -162.820, Y  +515.001, Z    +0.000, E1   -36.183, E3 +381632.880}
SPL {X  -162.820, Y  +520.482, Z    +0.000, E1   -36.096, E3 +381648.926}
SPL {X  -162.820, Y  +524.107, Z    +0.000, E1   -36.045, E3 +381659.510}
SPL {X  -162.820, Y  +527.962, Z    +0.000, E1   -36.074, E3 +381670.443}
SPL {X  -162.820, Y  +532.253, Z    +0.000, E1   -36.170, E3 +381682.032}
SPL {X  -162.820, Y  +536.031, Z    +0.000, E1   -36.058, E3 +381693.570}
SPL {X  -162.820, Y  +541.179, Z    +0.000, E1   -36.085, E3 +381708.210}
SPL {X  -162.820, Y  +546.355, Z    +0.000, E1   -36.114, E3 +381722.755}
SPL {X  -162.820, Y  +551.776, Z    +0.000, E1   -36.108, E3 +381738.389}
SPL {X  -162.820, Y  +556.944, Z    +0.000, E1   -36.118, E3 +381752.959}
SPL {X  -162.820, Y  +561.684, Z    +0.000, E1   -36.118, E3 +381766.551}
SPL {X  -162.820, Y  +566.500, Z    +0.000, E1   -36.073, E3 +381780.554}
SPL {X  -162.820, Y  +570.319, Z    +0.000, E1   -36.045, E3 +381791.582}
SPL {X  -162.820, Y  +573.265, Z    +0.000, E1   -36.071, E3 +381799.819}
SPL {X  -162.820, Y  +578.070, Z    +0.000, E1   -36.120, E3 +381813.500}
SPL {X  -162.820, Y  +582.838, Z    +0.000, E1   -36.064, E3 +381827.243}
SPL {X  -162.820, Y  +586.693, Z    +0.000, E1   -36.086, E3 +381838.219}
SPL {X  -162.820, Y  +590.250, Z    +0.000, E1   -36.075, E3 +381848.337}
SPL {X  -162.820, Y  +592.727, Z    +0.000, E1   -35.960, E3 +381856.162}
SPL {X  -162.820, Y  +597.399, Z    +0.000, E1   -36.147, E3 +381868.510}
SPL {X  -162.820, Y  +602.243, Z    +0.000, E1   -36.085, E3 +381882.656}
SPL {X  -162.820, Y  +606.975, Z    +0.000, E1   -36.102, E3 +381896.101}
SPL {X  -162.820, Y  +611.980, Z    +0.000, E1   -36.072, E3 +381910.647}
SPL {X  -162.820, Y  +616.897, Z    +0.000, E1   -36.061, E3 +381924.696}
SPL {X  -162.820, Y  +621.516, Z    +0.000, E1   -36.072, E3 +381937.895}
SPL {X  -162.820, Y  +626.243, Z    +0.000, E1   -36.105, E3 +381951.137}
SPL {X  -162.820, Y  +630.571, Z    +0.000, E1   -36.057, E3 +381963.839}
SPL {X  -162.820, Y  +635.505, Z    +0.000, E1   -36.079, E3 +381977.845}
SPL {X  -162.820, Y  +641.277, Z    +0.000, E1   -36.126, E3 +381994.138}
SPL {X  -162.820, Y  +646.320, Z    +0.000, E1   -36.078, E3 +382008.703}
SPL {X  -162.820, Y  +651.289, Z    +0.000, E1   -36.059, E3 +382023.159}
SPL {X  -162.820, Y  +656.677, Z    +0.000, E1   -36.110, E3 +382038.172}
SPL {X  -162.820, Y  +661.560, Z    +0.000, E1   -36.068, E3 +382052.435}
SPL {X  -162.820, Y  +666.386, Z    +0.000, E1   -36.048, E3 +382066.320}
SPL {X  -162.820, Y  +672.345, Z    +0.000, E1   -36.097, E3 +382083.260}
SPL {X  -162.761, Y  +677.889, Z    +0.000, E1   -36.122, E3 +382098.725}
SPL {X  -162.577, Y  +682.401, Z    +0.000, E1   -36.021, E3 +382112.342}
SPL {X  -162.187, Y  +687.846, Z    +0.000, E1   -36.007, E3 +382128.011}
SPL {X  -161.667, Y  +692.839, Z    +0.000, E1   -35.918, E3 +382142.776}
SPL {X  -161.078, Y  +697.256, Z    +0.000, E1   -35.797, E3 +382156.112}
SPL {X  -160.313, Y  +701.964, Z    +0.000, E1   -35.709, E3 +382170.187}
SPL {X  -159.317, Y  +707.091, Z    +0.000, E1   -35.482, E3 +382186.211}
SPL {X  -158.510, Y  +710.714, Z    +0.000, E1   -35.230, E3 +382197.922}
SPL {X  -155.037, Y  +723.239, Z    +0.000, E1   -39.382, E3 +382207.019}
SPL {X  -152.141, Y  +731.494, Z    +0.000, E1   -35.181, E3 +382265.824}
ENDSPLINE

SPLINE
SPL {X  -160.133, Y  +702.956, Z    +0.000, E1   -19.806, E3 +382309.362}
SPL {X  -161.979, Y  +690.023, Z    +0.000, E1   -12.991, E3 +382312.279}
SPL {X  -162.641, Y  +681.139, Z    +0.000, E1    -7.893, E3 +382314.371}
SPL {X  -162.815, Y  +674.833, Z    +0.000, E1    -4.093, E3 +382311.987}
SPL {X  -162.820, Y  +669.862, Z    +0.000, E1    -0.751, E3 +382315.205}
SPL {X  -162.820, Y  +665.790, Z    +0.000, E1    +2.338, E3 +382314.577}
SPL {X  -162.820, Y  +660.758, Z    +0.000, E1    +6.523, E3 +382314.678}
SPL {X  -162.820, Y  +650.583, Z    +0.000, E1   +16.035, E3 +382313.651}
SPL {X  -162.820, Y  +629.267, Z    +0.000, E1   +31.872, E3 +382324.799}
SPL {X  -162.820, Y  +617.390, Z    +0.000, E1   +35.413, E3 +382341.729}
SPL {X  -162.820, Y  +596.392, Z    +0.000, E1   +37.895, E3 +382382.469}
ENDSPLINE

SPLINE
SPL {X  -162.820, Y  +601.432, Z    +0.000, E1   +34.026, E3 +382391.767}
ENDSPLINE

SPLINE
SPL {X  -162.820, Y  +597.570, Z    +0.000, E1   +33.919, E3 +382404.664}
SPL {X  -162.820, Y  +592.692, Z    +0.000, E1   +33.779, E3 +382420.556}
SPL {X  -162.820, Y  +588.795, Z    +0.000, E1   +33.876, E3 +382431.993}
SPL {X  -162.820, Y  +585.519, Z    +0.000, E1   +33.888, E3 +382442.078}
SPL {X  -162.820, Y  +582.066, Z    +0.000, E1   +33.857, E3 +382453.012}
SPL {X  -162.820, Y  +577.919, Z    +0.000, E1   +33.841, E3 +382466.065}
SPL {X  -162.820, Y  +573.566, Z    +0.000, E1   +33.899, E3 +382479.140}
SPL {X  -162.820, Y  +569.298, Z    +0.000, E1   +33.851, E3 +382492.781}
SPL {X  -162.820, Y  +563.983, Z    +0.000, E1   +33.916, E3 +382508.922}
SPL {X  -162.820, Y  +559.395, Z    +0.000, E1   +33.796, E3 +382523.803}
SPL {X  -162.820, Y  +554.453, Z    +0.000, E1   +33.841, E3 +382539.028}
SPL {X  -162.820, Y  +549.726, Z    +0.000, E1   +33.905, E3 +382553.131}
SPL {X  -162.820, Y  +545.760, Z    +0.000, E1   +33.901, E3 +382565.527}
SPL {X  -162.820, Y  +541.668, Z    +0.000, E1   +33.787, E3 +382578.927}
SPL {X  -162.820, Y  +537.061, Z    +0.000, E1   +33.897, E3 +382592.586}
SPL {X  -162.820, Y  +532.164, Z    +0.000, E1   +33.861, E3 +382608.059}
SPL {X  -162.820, Y  +528.475, Z    +0.000, E1   +33.876, E3 +382619.228}
SPL {X  -162.820, Y  +524.900, Z    +0.000, E1   +33.820, E3 +382630.887}
SPL {X  -162.820, Y  +520.532, Z    +0.000, E1   +33.805, E3 +382644.454}
SPL {X  -162.820, Y  +516.814, Z    +0.000, E1   +33.917, E3 +382655.290}
SPL {X  -162.820, Y  +512.685, Z    +0.000, E1   +33.830, E3 +382668.733}
SPL {X  -162.820, Y  +508.888, Z    +0.000, E1   +33.871, E3 +382680.148}
SPL {X  -162.820, Y  +505.651, Z    +0.000, E1   +33.839, E3 +382690.465}
SPL {X  -162.820, Y  +500.931, Z    +0.000, E1   +34.256, E3 +382702.338}
SPL {X  -162.820, Y  +481.122, Z    +0.000, E1   +41.279, E3 +382712.603}
SPL {X  -162.820, Y  +477.698, Z    +0.000, E1   +40.353, E3 +382726.659}
SPL {X  -162.820, Y  +474.538, Z    +0.000, E1   +39.267, E3 +382740.834}
SPL {X  -162.820, Y  +472.097, Z    +0.000, E1   +38.411, E3 +382752.378}
SPL {X  -162.820, Y  +469.308, Z    +0.000, E1   +37.839, E3 +382763.182}
SPL {X  -162.820, Y  +467.216, Z    +0.000, E1   +37.215, E3 +382772.749}
SPL {X  -162.820, Y  +462.598, Z    +0.000, E1   +37.325, E3 +382784.703}
SPL {X  -162.820, Y  +457.832, Z    +0.000, E1   +37.294, E3 +382797.989}
SPL {X  -162.820, Y  +452.986, Z    +0.000, E1   +37.368, E3 +382810.723}
SPL {X  -162.820, Y  +447.084, Z    +0.000, E1   +37.389, E3 +382826.914}
SPL {X  -162.820, Y  +440.036, Z    +0.000, E1   +37.326, E3 +382846.532}
SPL {X  -162.820, Y  +434.320, Z    +0.000, E1   +37.343, E3 +382861.855}
SPL {X  -162.820, Y  +430.091, Z    +0.000, E1   +37.424, E3 +382872.855}
SPL {X  -162.820, Y  +426.177, Z    +0.000, E1   +37.250, E3 +382884.678}
SPL {X  -162.820, Y  +421.391, Z    +0.000, E1   +37.346, E3 +382897.142}
SPL {X  -162.820, Y  +416.811, Z    +0.000, E1   +37.348, E3 +382909.676}
SPL {X  -162.820, Y  +411.860, Z    +0.000, E1   +37.402, E3 +382922.828}
SPL {X  -162.820, Y  +407.726, Z    +0.000, E1   +37.291, E3 +382934.775}
SPL {X  -162.820, Y  +403.543, Z    +0.000, E1   +37.305, E3 +382946.121}
SPL {X  -162.820, Y  +399.300, Z    +0.000, E1   +37.355, E3 +382957.405}
SPL {X  -162.820, Y  +395.182, Z    +0.000, E1   +37.347, E3 +382968.694}
SPL {X  -162.820, Y  +390.797, Z    +0.000, E1   +37.358, E3 +382980.606}
SPL {X  -162.820, Y  +386.671, Z    +0.000, E1   +37.363, E3 +382991.787}
SPL {X  -162.820, Y  +382.174, Z    +0.000, E1   +37.329, E3 +383004.365}
SPL {X  -162.785, Y  +377.133, Z    +0.000, E1   +37.299, E3 +383018.294}
SPL {X  -162.623, Y  +372.484, Z    +0.000, E1   +37.337, E3 +383030.734}
SPL {X  -162.331, Y  +367.894, Z    +0.000, E1   +37.251, E3 +383043.846}
SPL {X  -161.920, Y  +363.407, Z    +0.000, E1   +37.164, E3 +383056.580}
SPL {X  -161.341, Y  +358.603, Z    +0.000, E1   +37.117, E3 +383070.061}
SPL {X  -160.616, Y  +353.801, Z    +0.000, E1   +36.942, E3 +383084.225}
SPL {X  -159.837, Y  +349.474, Z    +0.000, E1   +36.824, E3 +383096.669}
SPL {X  -158.862, Y  +344.820, Z    +0.000, E1   +36.732, E3 +383110.032}
SPL {X  -157.959, Y  +341.011, Z    +0.000, E1   +36.448, E3 +383121.929}
SPL {X  -154.495, Y  +329.104, Z    +0.000, E1   +40.891, E3 +383126.811}
SPL {X  -152.543, Y  +323.569, Z    +0.000, E1   +41.772, E3 +383134.568}
SPL {X  -150.942, Y  +319.452, Z    +0.000, E1   +36.529, E3 +383187.118}
ENDSPLINE

SPLINE
SPL {X  -159.264, Y  +346.659, Z    +0.000, E1   +22.083, E3 +383227.692}
SPL {X  -161.245, Y  +357.907, Z    +0.000, E1   +16.095, E3 +383241.125}
SPL {X  -162.697, Y  +374.161, Z    +0.000, E1    +7.119, E3 +383239.114}
SPL {X  -162.820, Y  +380.878, Z    +0.000, E1    +2.854, E3 +383241.946}
SPL {X  -162.820, Y  +385.313, Z    +0.000, E1    -0.228, E3 +383241.726}
SPL {X  -162.820, Y  +389.965, Z    +0.000, E1    -3.918, E3 +383241.094}
SPL {X  -162.820, Y  +394.532, Z    +0.000, E1    -7.849, E3 +383242.642}
SPL {X  -162.820, Y  +400.765, Z    +0.000, E1   -14.108, E3 +383240.109}
SPL {X  -162.820, Y  +411.829, Z    +0.000, E1   -24.195, E3 +383242.187}
SPL {X  -162.820, Y  +434.900, Z    +0.000, E1   -34.666, E3 +383269.551}
SPL {X  -162.820, Y  +465.440, Z    +0.000, E1   -41.264, E3 +383310.859}
ENDSPLINE

SPLINE
SPL {X  -162.820, Y  +460.175, Z    +0.000, E1   -36.098, E3 +383328.659}
ENDSPLINE

